LIN {X 0,Y 369.974,Z 1121.521,A -85,B 0,C 180,E1 18072.043,E2 18072.043} C_VEL
LIN {X 0,Y 371.684,Z 1112.764,A -85,B 0,C 180,E1 18068.54,E2 18068.54} C_VEL
LIN {X 0,Y 373.899,Z 1103.179,A -85,B 0,C 180,E1 18065.344,E2 18065.344} C_VEL
LIN {X 0,Y 376.935,Z 1091.306,A -85,B 0,C 180,E1 18062.045,E2 18062.045} C_VEL
LIN {X 0,Y 380.529,Z 1078.476,A -85,B 0,C 180,E1 18059.003,E2 18059.003} C_VEL
LIN {X 0,Y 384.517,Z 1064.377,A -85,B 0,C 180,E1 18056.189,E2 18056.189} C_VEL
LIN {X 0,Y 389.236,Z 1048.185,A -85,B 0,C 180,E1 18053.419,E2 18053.419} C_VEL
LIN {X 0,Y 393.672,Z 1032.569,A -85,B 0,C 180,E1 18051.146,E2 18051.146} C_VEL
LIN {X 0,Y 399.011,Z 1013.125,A -85,B 0,C 180,E1 18048.743,E2 18048.743} C_VEL
LIN {X 0,Y 403.673,Z 995.222,A -85,B 0,C 180,E1 18046.873,E2 18046.873} C_VEL
LIN {X 0,Y 408.313,Z 975.608,A -85,B 0,C 180,E1 18045.151,E2 18045.151} C_VEL
LIN {X 0,Y 412.424,Z 956.575,A -85,B 0,C 180,E1 18043.742,E2 18043.742} C_VEL
LIN {X 0,Y 416.471,Z 934.827,A -85,B 0,C 180,E1 18042.425,E2 18042.425} C_VEL
LIN {X 0,Y 419.947,Z 913.057,A -85,B 0,C 180,E1 18041.359,E2 18041.359} C_VEL
LIN {X 0,Y 422.727,Z 890.385,A -85,B 0,C 180,E1 18040.517,E2 18040.517} C_VEL
LIN {X 0,Y 424.934,Z 866.356,A -85,B 0,C 180,E1 18039.872,E2 18039.872} C_VEL
LIN {X 0,Y 433.354,Z 685.979,A -85,B 0,C 180,E1 18036.447,E2 18036.447} C_VEL
LIN {X 0,Y 436.488,Z 620.977,A -85,B 0,C 180,E1 18035.218,E2 18035.218} C_VEL
LIN {X 0,Y 425.983,Z 605.601,A -85,B 0,C 180,E1 18032.674,E2 18032.674} C_VEL
LIN {X 0,Y 417.336,Z 593.961,A -85,B 0,C 180,E1 18030.366,E2 18030.366} C_VEL
LIN {X 0,Y 410.196,Z 584.627,A -85,B 0,C 180,E1 18028.261,E2 18028.261} C_VEL
LIN {X 0,Y 406.17,Z 579.545,A -85,B 0,C 180,E1 18026.98,E2 18026.98} C_VEL
LIN {X 0,Y 402.194,Z 574.58,A -85,B 0,C 180,E1 18025.631,E2 18025.631} C_VEL
LIN {X 0,Y 398.427,Z 569.939,A -85,B 0,C 180,E1 18024.264,E2 18024.264} C_VEL
LIN {X 0,Y 393.864,Z 564.736,A -85,B 0,C 180,E1 18022.484,E2 18022.484} C_VEL
LIN {X 0,Y 392.693,Z 563.037,A -85,B 0,C 180,E1 18021.98,E2 18021.98} C_VEL
LIN {X 0,Y 389.293,Z 559.846,A -85,B 0,C 180,E1 18020.523,E2 18020.523} C_VEL
LIN {X 0,Y 387.428,Z 556.914,A -85,B 0,C 180,E1 18019.603,E2 18019.603} C_VEL
LIN {X 0,Y 384.221,Z 554.346,A -85,B 0,C 180,E1 18018.04,E2 18018.04} C_VEL
LIN {X 0,Y 382.022,Z 550.476,A -85,B 0,C 180,E1 18016.733,E2 18016.733} C_VEL
LIN {X 0,Y 378.428,Z 548.236,A -85,B 0,C 180,E1 18014.615,E2 18014.615} C_VEL
LIN {X 0,Y 376.464,Z 544.941,A -85,B 0,C 180,E1 18013.126,E2 18013.126} C_VEL
LIN {X 0,Y 376.048,Z 543.83,A -85,B 0,C 180,E1 18012.75,E2 18012.75} C_VEL
LIN {X 0,Y 372.297,Z 541.914,A -85,B 0,C 180,E1 18009.585,E2 18009.585} C_VEL
LIN {X 0,Y 370.014,Z 538.337,A -85,B 0,C 180,E1 18006.517,E2 18006.517} C_VEL
LIN {X 0,Y 369.746,Z 536.98,A -85,B 0,C 180,E1 18005.743,E2 18005.743} C_VEL
LIN {X 0,Y 369.744,Z 536.974,A -85,B 0,C 180,E1 18001.55,E2 18001.55} C_VEL
LIN {X 0,Y 369.74,Z 536.973,A -85,B 0,C 180,E1 17997.521,E2 17997.521} C_VEL
LIN {X 0,Y 369.757,Z 537.107,A -85,B 0,C 180,E1 17994.57,E2 17994.57} C_VEL
LIN {X 0,Y 370.779,Z 540.029,A -85,B 0,C 180,E1 17992.719,E2 17992.719} C_VEL
LIN {X 0,Y 373.759,Z 542.916,A -85,B 0,C 180,E1 17989.519,E2 17989.519} C_VEL
LIN {X 0,Y 376.203,Z 544.056,A -85,B 0,C 180,E1 17987.608,E2 17987.608} C_VEL
LIN {X 0,Y 377.601,Z 547.177,A -85,B 0,C 180,E1 17986.448,E2 17986.448} C_VEL
LIN {X 0,Y 380.461,Z 549.827,A -85,B 0,C 180,E1 17984.608,E2 17984.608} C_VEL
LIN {X 0,Y 382.158,Z 550.727,A -85,B 0,C 180,E1 17983.665,E2 17983.665} C_VEL
LIN {X 0,Y 384.245,Z 554.349,A -85,B 0,C 180,E1 17982.432,E2 17982.432} C_VEL
LIN {X 0,Y 387.893,Z 557.427,A -85,B 0,C 180,E1 17980.657,E2 17980.657} C_VEL
LIN {X 0,Y 390.551,Z 561.348,A -85,B 0,C 180,E1 17979.39,E2 17979.39} C_VEL
LIN {X 0,Y 393.287,Z 563.765,A -85,B 0,C 180,E1 17978.251,E2 17978.251} C_VEL
LIN {X 0,Y 396.379,Z 567.873,A -85,B 0,C 180,E1 17976.985,E2 17976.985} C_VEL
LIN {X 0,Y 398.446,Z 569.988,A -85,B 0,C 180,E1 17976.21,E2 17976.21} C_VEL
LIN {X 0,Y 406.022,Z 579.905,A -85,B 0,C 180,E1 17973.531,E2 17973.531} C_VEL
LIN {X 0,Y 413.975,Z 590.853,A -85,B 0,C 180,E1 17971.036,E2 17971.036} C_VEL
LIN {X 0,Y 422.851,Z 603.946,A -85,B 0,C 180,E1 17968.536,E2 17968.536} C_VEL
LIN {X 0,Y 431.125,Z 616.822,A -85,B 0,C 180,E1 17966.419,E2 17966.419} C_VEL
LIN {X 0,Y 436.595,Z 626.032,A -85,B 0,C 180,E1 17965.103,E2 17965.103} C_VEL
LIN {X 0,Y 426.617,Z 841.95,A -85,B 0,C 180,E1 17961.024,E2 17961.024} C_VEL
LIN {X 0,Y 424.207,Z 890.642,A -85,B 0,C 180,E1 17960.077,E2 17960.077} C_VEL
LIN {X 0,Y 421.841,Z 913.593,A -85,B 0,C 180,E1 17959.447,E2 17959.447} C_VEL
LIN {X 0,Y 418.914,Z 935.594,A -85,B 0,C 180,E1 17958.636,E2 17958.636} C_VEL
LIN {X 0,Y 415.455,Z 956.499,A -85,B 0,C 180,E1 17957.633,E2 17957.633} C_VEL
LIN {X 0,Y 411.316,Z 978.245,A -85,B 0,C 180,E1 17956.341,E2 17956.341} C_VEL
LIN {X 0,Y 407.088,Z 997.769,A -85,B 0,C 180,E1 17954.921,E2 17954.921} C_VEL
LIN {X 0,Y 402.036,Z 1019.156,A -85,B 0,C 180,E1 17953.053,E2 17953.053} C_VEL
LIN {X 0,Y 397.539,Z 1036.83,A -85,B 0,C 180,E1 17951.221,E2 17951.221} C_VEL
LIN {X 0,Y 392.445,Z 1055.81,A -85,B 0,C 180,E1 17948.904,E2 17948.904} C_VEL
LIN {X 0,Y 387.77,Z 1073.02,A -85,B 0,C 180,E1 17946.44,E2 17946.44} C_VEL
LIN {X 0,Y 383.358,Z 1088.948,A -85,B 0,C 180,E1 17943.748,E2 17943.748} C_VEL
LIN {X 0,Y 379.505,Z 1103.464,A -85,B 0,C 180,E1 17940.914,E2 17940.914} C_VEL
LIN {X 0,Y 376.133,Z 1116.554,A -85,B 0,C 180,E1 17937.895,E2 17937.895} C_VEL
LIN {X 0,Y 373.235,Z 1129.035,A -85,B 0,C 180,E1 17934.534,E2 17934.534} C_VEL
LIN {X 0,Y 371.275,Z 1138.569,A -85,B 0,C 180,E1 17931.484,E2 17931.484} C_VEL
LIN {X 0,Y 369.619,Z 1148.226,A -85,B 0,C 180,E1 17927.789,E2 17927.789} C_VEL
LIN {X 0,Y 368.729,Z 1154.956,A -85,B 0,C 180,E1 17924.606,E2 17924.606} C_VEL
LIN {X 0,Y 368.194,Z 1161.002,A -85,B 0,C 180,E1 17920.958,E2 17920.958} C_VEL
LIN {X 0,Y 367.999,Z 1164.643,A -85,B 0,C 180,E1 17917.965,E2 17917.965} C_VEL
LIN {X 0,Y 367.927,Z 1167.483,A -85,B 0,C 180,E1 17914.52,E2 17914.52} C_VEL
LIN {X 0,Y 367.923,Z 1168.636,A -85,B 0,C 180,E1 17911.245,E2 17911.245} C_VEL
LIN {X 0,Y 367.926,Z 1168.565,A -85,B 0,C 180,E1 17908.287,E2 17908.287} C_VEL
LIN {X 0,Y 367.93,Z 1167.053,A -85,B 0,C 180,E1 17904.855,E2 17904.855} C_VEL
LIN {X 0,Y 368.013,Z 1164.312,A -85,B 0,C 180,E1 17901.72,E2 17901.72} C_VEL
LIN {X 0,Y 368.272,Z 1159.89,A -85,B 0,C 180,E1 17898.251,E2 17898.251} C_VEL
LIN {X 0,Y 368.841,Z 1154.02,A -85,B 0,C 180,E1 17894.915,E2 17894.915} C_VEL
LIN {X 0,Y 369.869,Z 1146.741,A -85,B 0,C 180,E1 17891.561,E2 17891.561} C_VEL
LIN {X 0,Y 371.46,Z 1137.631,A -85,B 0,C 180,E1 17888.194,E2 17888.194} C_VEL
LIN {X 0,Y 373.736,Z 1126.85,A -85,B 0,C 180,E1 17884.825,E2 17884.825} C_VEL
LIN {X 0,Y 376.617,Z 1114.607,A -85,B 0,C 180,E1 17881.626,E2 17881.626} C_VEL
LIN {X 0,Y 380.345,Z 1100.097,A -85,B 0,C 180,E1 17878.4,E2 17878.4} C_VEL
LIN {X 0,Y 384.323,Z 1085.496,A -85,B 0,C 180,E1 17875.628,E2 17875.628} C_VEL
LIN {X 0,Y 388.891,Z 1068.742,A -85,B 0,C 180,E1 17872.921,E2 17872.921} C_VEL
LIN {X 0,Y 393.728,Z 1051.242,A -85,B 0,C 180,E1 17870.495,E2 17870.495} C_VEL
LIN {X 0,Y 398.569,Z 1032.731,A -85,B 0,C 180,E1 17868.334,E2 17868.334} C_VEL
LIN {X 0,Y 403.725,Z 1012.106,A -85,B 0,C 180,E1 17866.293,E2 17866.293} C_VEL
LIN {X 0,Y 408.111,Z 993.164,A -85,B 0,C 180,E1 17864.724,E2 17864.724} C_VEL
LIN {X 0,Y 412.553,Z 971.99,A -85,B 0,C 180,E1 17863.266,E2 17863.266} C_VEL
LIN {X 0,Y 416.147,Z 952.514,A -85,B 0,C 180,E1 17862.164,E2 17862.164} C_VEL
LIN {X 0,Y 419.778,Z 929.35,A -85,B 0,C 180,E1 17861.118,E2 17861.118} C_VEL
LIN {X 0,Y 422.268,Z 909.791,A -85,B 0,C 180,E1 17860.439,E2 17860.439} C_VEL
LIN {X 0,Y 424.551,Z 884.65,A -85,B 0,C 180,E1 17859.8,E2 17859.8} C_VEL
LIN {X 0,Y 433.122,Z 697.721,A -85,B 0,C 180,E1 17856.257,E2 17856.257} C_VEL
LIN {X 0,Y 436.44,Z 625.581,A -85,B 0,C 180,E1 17854.869,E2 17854.869} C_VEL
LIN {X 0,Y 425.319,Z 607.642,A -85,B 0,C 180,E1 17852.132,E2 17852.132} C_VEL
LIN {X 0,Y 415.18,Z 592.599,A -85,B 0,C 180,E1 17849.345,E2 17849.345} C_VEL
LIN {X 0,Y 407.907,Z 582.585,A -85,B 0,C 180,E1 17847.124,E2 17847.124} C_VEL
LIN {X 0,Y 403.893,Z 577.15,A -85,B 0,C 180,E1 17845.79,E2 17845.79} C_VEL
LIN {X 0,Y 400.129,Z 572.41,A -85,B 0,C 180,E1 17844.467,E2 17844.467} C_VEL
LIN {X 0,Y 397.545,Z 568.885,A -85,B 0,C 180,E1 17843.493,E2 17843.493} C_VEL
LIN {X 0,Y 394.054,Z 565.064,A -85,B 0,C 180,E1 17842.135,E2 17842.135} C_VEL
LIN {X 0,Y 392.77,Z 563.107,A -85,B 0,C 180,E1 17841.582,E2 17841.582} C_VEL
LIN {X 0,Y 389.424,Z 560.029,A -85,B 0,C 180,E1 17840.163,E2 17840.163} C_VEL
LIN {X 0,Y 387.637,Z 556.986,A -85,B 0,C 180,E1 17839.278,E2 17839.278} C_VEL
LIN {X 0,Y 384.248,Z 554.358,A -85,B 0,C 180,E1 17837.646,E2 17837.646} C_VEL
LIN {X 0,Y 382.144,Z 550.727,A -85,B 0,C 180,E1 17836.414,E2 17836.414} C_VEL
LIN {X 0,Y 378.187,Z 547.968,A -85,B 0,C 180,E1 17834.077,E2 17834.077} C_VEL
LIN {X 0,Y 376.387,Z 544.727,A -85,B 0,C 180,E1 17832.698,E2 17832.698} C_VEL
LIN {X 0,Y 376.11,Z 543.795,A -85,B 0,C 180,E1 17832.435,E2 17832.435} C_VEL
LIN {X 0,Y 372.136,Z 541.73,A -85,B 0,C 180,E1 17829.121,E2 17829.121} C_VEL
LIN {X 0,Y 370.12,Z 538.604,A -85,B 0,C 180,E1 17826.514,E2 17826.514} C_VEL
LIN {X 0,Y 369.739,Z 536.974,A -85,B 0,C 180,E1 17825.586,E2 17825.586} C_VEL
LIN {X 0,Y 369.738,Z 536.977,A -85,B 0,C 180,E1 17821.394,E2 17821.394} C_VEL
LIN {X 0,Y 369.729,Z 536.982,A -85,B 0,C 180,E1 17817.365,E2 17817.365} C_VEL
LIN {X 0,Y 369.766,Z 537.211,A -85,B 0,C 180,E1 17813.634,E2 17813.634} C_VEL
LIN {X 0,Y 370.756,Z 539.978,A -85,B 0,C 180,E1 17811.938,E2 17811.938} C_VEL
LIN {X 0,Y 373.997,Z 543.047,A -85,B 0,C 180,E1 17808.589,E2 17808.589} C_VEL
LIN {X 0,Y 376.203,Z 544.103,A -85,B 0,C 180,E1 17806.904,E2 17806.904} C_VEL
LIN {X 0,Y 377.726,Z 547.39,A -85,B 0,C 180,E1 17805.67,E2 17805.67} C_VEL
LIN {X 0,Y 380.657,Z 549.896,A -85,B 0,C 180,E1 17803.833,E2 17803.833} C_VEL
LIN {X 0,Y 382.168,Z 550.759,A -85,B 0,C 180,E1 17803,E2 17803} C_VEL
LIN {X 0,Y 384.353,Z 554.514,A -85,B 0,C 180,E1 17801.723,E2 17801.723} C_VEL
LIN {X 0,Y 387.868,Z 557.472,A -85,B 0,C 180,E1 17800.028,E2 17800.028} C_VEL
LIN {X 0,Y 390.55,Z 561.329,A -85,B 0,C 180,E1 17798.761,E2 17798.761} C_VEL
LIN {X 0,Y 393.217,Z 563.653,A -85,B 0,C 180,E1 17797.657,E2 17797.657} C_VEL
LIN {X 0,Y 396.404,Z 567.901,A -85,B 0,C 180,E1 17796.356,E2 17796.356} C_VEL
LIN {X 0,Y 398.392,Z 569.905,A -85,B 0,C 180,E1 17795.616,E2 17795.616} C_VEL
LIN {X 0,Y 402.071,Z 574.487,A -85,B 0,C 180,E1 17794.282,E2 17794.282} C_VEL
LIN {X 0,Y 403.96,Z 576.86,A -85,B 0,C 180,E1 17793.63,E2 17793.63} C_VEL
LIN {X 0,Y 408.347,Z 582.296,A -85,B 0,C 180,E1 17792.196,E2 17792.196} C_VEL
LIN {X 0,Y 412.91,Z 588.21,A -85,B 0,C 180,E1 17790.795,E2 17790.795} C_VEL
LIN {X 0,Y 420.03,Z 597.504,A -85,B 0,C 180,E1 17788.779,E2 17788.779} C_VEL
LIN {X 0,Y 430.409,Z 611.995,A -85,B 0,C 180,E1 17786.115,E2 17786.115} C_VEL
LIN {X 0,Y 436.464,Z 621.114,A -85,B 0,C 180,E1 17784.679,E2 17784.679} C_VEL
LIN {X 0,Y 426.709,Z 829.94,A -85,B 0,C 180,E1 17780.74,E2 17780.74} C_VEL
LIN {X 0,Y 424.596,Z 870.779,A -85,B 0,C 180,E1 17779.937,E2 17779.937} C_VEL
LIN {X 0,Y 422.391,Z 893.197,A -85,B 0,C 180,E1 17779.296,E2 17779.296} C_VEL
LIN {X 0,Y 419.347,Z 916.813,A -85,B 0,C 180,E1 17778.374,E2 17778.374} C_VEL
LIN {X 0,Y 416.239,Z 936.052,A -85,B 0,C 180,E1 17777.414,E2 17777.414} C_VEL
LIN {X 0,Y 411.993,Z 958.492,A -85,B 0,C 180,E1 17776.03,E2 17776.03} C_VEL
LIN {X 0,Y 408.091,Z 976.509,A -85,B 0,C 180,E1 17774.683,E2 17774.683} C_VEL
LIN {X 0,Y 403.076,Z 997.396,A -85,B 0,C 180,E1 17772.819,E2 17772.819} C_VEL
LIN {X 0,Y 398.419,Z 1015.308,A -85,B 0,C 180,E1 17770.92,E2 17770.92} C_VEL
LIN {X 0,Y 393.512,Z 1033.103,A -85,B 0,C 180,E1 17768.687,E2 17768.687} C_VEL
LIN {X 0,Y 388.822,Z 1049.667,A -85,B 0,C 180,E1 17766.26,E2 17766.26} C_VEL
LIN {X 0,Y 384.391,Z 1064.772,A -85,B 0,C 180,E1 17763.646,E2 17763.646} C_VEL
LIN {X 0,Y 380.431,Z 1078.817,A -85,B 0,C 180,E1 17760.831,E2 17760.831} C_VEL
LIN {X 0,Y 378.216,Z 1086.719,A -85,B 0,C 180,E1 17759.02,E2 17759.02} C_VEL
LIN {X 0,Y 376.201,Z 1090.945,A -85,B 0,C 180,E1 17758.078,E2 17758.078} C_VEL
LIN {X 0,Y 367.563,Z 1101.74,A -85,B 0,C 180,E1 17755.588,E2 17755.588} C_VEL
LIN {X 0,Y 366.052,Z 1104.763,A -85,B 0,C 180,E1 17754.692,E2 17754.692} C_VEL
LIN {X 0,Y 363.781,Z 1114.173,A -85,B 0,C 180,E1 17751.442,E2 17751.442} C_VEL
LIN {X 0,Y 362.006,Z 1122.695,A -85,B 0,C 180,E1 17747.854,E2 17747.854} C_VEL
LIN {X 0,Y 360.934,Z 1129.295,A -85,B 0,C 180,E1 17744.438,E2 17744.438} C_VEL
LIN {X 0,Y 360.309,Z 1134.534,A -85,B 0,C 180,E1 17740.877,E2 17740.877} C_VEL
LIN {X 0,Y 360.035,Z 1138.029,A -85,B 0,C 180,E1 17737.661,E2 17737.661} C_VEL
LIN {X 0,Y 359.946,Z 1140.516,A -85,B 0,C 180,E1 17733.982,E2 17733.982} C_VEL
LIN {X 0,Y 359.922,Z 1141.386,A -85,B 0,C 180,E1 17730.955,E2 17730.955} C_VEL
LIN {X 0,Y 359.937,Z 1141.148,A -85,B 0,C 180,E1 17727.453,E2 17727.453} C_VEL
LIN {X 0,Y 359.967,Z 1139.462,A -85,B 0,C 180,E1 17724.101,E2 17724.101} C_VEL
LIN {X 0,Y 360.154,Z 1136.572,A -85,B 0,C 180,E1 17720.734,E2 17720.734} C_VEL
LIN {X 0,Y 360.579,Z 1131.982,A -85,B 0,C 180,E1 17717.183,E2 17717.183} C_VEL
LIN {X 0,Y 361.415,Z 1126.219,A -85,B 0,C 180,E1 17713.775,E2 17713.775} C_VEL
LIN {X 0,Y 362.854,Z 1118.465,A -85,B 0,C 180,E1 17710.188,E2 17710.188} C_VEL
LIN {X 0,Y 364.909,Z 1109.488,A -85,B 0,C 180,E1 17706.761,E2 17706.761} C_VEL
LIN {X 0,Y 367.708,Z 1098.548,A -85,B 0,C 180,E1 17703.342,E2 17703.342} C_VEL
LIN {X 0,Y 371.189,Z 1086.365,A -85,B 0,C 180,E1 17700.111,E2 17700.111} C_VEL
LIN {X 0,Y 374.999,Z 1073.488,A -85,B 0,C 180,E1 17697.231,E2 17697.231} C_VEL
LIN {X 0,Y 379.793,Z 1057.789,A -85,B 0,C 180,E1 17694.236,E2 17694.236} C_VEL
LIN {X 0,Y 384.442,Z 1042.497,A -85,B 0,C 180,E1 17691.758,E2 17691.758} C_VEL
LIN {X 0,Y 389.665,Z 1024.824,A -85,B 0,C 180,E1 17689.326,E2 17689.326} C_VEL
LIN {X 0,Y 394.549,Z 1007.564,A -85,B 0,C 180,E1 17687.3,E2 17687.3} C_VEL
LIN {X 0,Y 399.514,Z 988.481,A -85,B 0,C 180,E1 17685.412,E2 17685.412} C_VEL
LIN {X 0,Y 404.278,Z 968.766,A -85,B 0,C 180,E1 17683.766,E2 17683.766} C_VEL
LIN {X 0,Y 408.611,Z 948.141,A -85,B 0,C 180,E1 17682.355,E2 17682.355} C_VEL
LIN {X 0,Y 412.602,Z 926.618,A -85,B 0,C 180,E1 17681.146,E2 17681.146} C_VEL
LIN {X 0,Y 415.736,Z 905.591,A -85,B 0,C 180,E1 17680.218,E2 17680.218} C_VEL
LIN {X 0,Y 418.471,Z 882.758,A -85,B 0,C 180,E1 17679.442,E2 17679.442} C_VEL
LIN {X 0,Y 420.221,Z 860.799,A -85,B 0,C 180,E1 17678.912,E2 17678.912} C_VEL
LIN {X 0,Y 429.901,Z 661.299,A -85,B 0,C 180,E1 17675.114,E2 17675.114} C_VEL
LIN {X 0,Y 431.671,Z 625.138,A -85,B 0,C 180,E1 17674.414,E2 17674.414} C_VEL
LIN {X 0,Y 422.321,Z 611.429,A -85,B 0,C 180,E1 17672.068,E2 17672.068} C_VEL
LIN {X 0,Y 414.179,Z 600.251,A -85,B 0,C 180,E1 17669.822,E2 17669.822} C_VEL
LIN {X 0,Y 407.276,Z 591.159,A -85,B 0,C 180,E1 17667.725,E2 17667.725} C_VEL
LIN {X 0,Y 403.607,Z 586.459,A -85,B 0,C 180,E1 17666.522,E2 17666.522} C_VEL
LIN {X 0,Y 399.717,Z 581.583,A -85,B 0,C 180,E1 17665.166,E2 17665.166} C_VEL
LIN {X 0,Y 395.235,Z 576.057,A -85,B 0,C 180,E1 17663.481,E2 17663.481} C_VEL
LIN {X 0,Y 391.616,Z 571.678,A -85,B 0,C 180,E1 17662.005,E2 17662.005} C_VEL
LIN {X 0,Y 390.571,Z 570.382,A -85,B 0,C 180,E1 17661.553,E2 17661.553} C_VEL
LIN {X 0,Y 387.196,Z 566.895,A -85,B 0,C 180,E1 17660.048,E2 17660.048} C_VEL
LIN {X 0,Y 385.874,Z 564.637,A -85,B 0,C 180,E1 17659.37,E2 17659.37} C_VEL
LIN {X 0,Y 382.582,Z 561.89,A -85,B 0,C 180,E1 17657.726,E2 17657.726} C_VEL
LIN {X 0,Y 380.276,Z 558.156,A -85,B 0,C 180,E1 17656.34,E2 17656.34} C_VEL
LIN {X 0,Y 376.808,Z 555.68,A -85,B 0,C 180,E1 17654.209,E2 17654.209} C_VEL
LIN {X 0,Y 374.843,Z 552.084,A -85,B 0,C 180,E1 17652.635,E2 17652.635} C_VEL
LIN {X 0,Y 374.274,Z 551.558,A -85,B 0,C 180,E1 17652.184,E2 17652.184} C_VEL
LIN {X 0,Y 370.628,Z 549.247,A -85,B 0,C 180,E1 17648.846,E2 17648.846} C_VEL
LIN {X 0,Y 368.792,Z 545.751,A -85,B 0,C 180,E1 17646.07,E2 17646.07} C_VEL
LIN {X 0,Y 368.514,Z 544.882,A -85,B 0,C 180,E1 17645.45,E2 17645.45} C_VEL
LIN {X 0,Y 367.489,Z 544.65,A -85,B 0,C 180,E1 17637.349,E2 17637.349} C_VEL
LIN {X 0,Y 368.674,Z 545.169,A -85,B 0,C 180,E1 17634.71,E2 17634.71} C_VEL
LIN {X 0,Y 370.02,Z 548.462,A -85,B 0,C 180,E1 17632.392,E2 17632.392} C_VEL
LIN {X 0,Y 373.522,Z 551.238,A -85,B 0,C 180,E1 17628.888,E2 17628.888} C_VEL
LIN {X 0,Y 374.781,Z 551.857,A -85,B 0,C 180,E1 17627.912,E2 17627.912} C_VEL
LIN {X 0,Y 376.512,Z 555.301,A -85,B 0,C 180,E1 17626.486,E2 17626.486} C_VEL
LIN {X 0,Y 379.513,Z 557.837,A -85,B 0,C 180,E1 17624.569,E2 17624.569} C_VEL
LIN {X 0,Y 380.599,Z 558.552,A -85,B 0,C 180,E1 17623.949,E2 17623.949} C_VEL
LIN {X 0,Y 383.003,Z 562.351,A -85,B 0,C 180,E1 17622.53,E2 17622.53} C_VEL
LIN {X 0,Y 386.169,Z 565.122,A -85,B 0,C 180,E1 17620.96,E2 17620.96} C_VEL
LIN {X 0,Y 388.957,Z 569.05,A -85,B 0,C 180,E1 17619.616,E2 17619.616} C_VEL
LIN {X 0,Y 391.401,Z 571.327,A -85,B 0,C 180,E1 17618.574,E2 17618.574} C_VEL
LIN {X 0,Y 394.72,Z 575.585,A -85,B 0,C 180,E1 17617.198,E2 17617.198} C_VEL
LIN {X 0,Y 396.397,Z 577.418,A -85,B 0,C 180,E1 17616.553,E2 17616.553} C_VEL
LIN {X 0,Y 403.575,Z 586.93,A -85,B 0,C 180,E1 17613.952,E2 17613.952} C_VEL
LIN {X 0,Y 411.399,Z 597.894,A -85,B 0,C 180,E1 17611.434,E2 17611.434} C_VEL
LIN {X 0,Y 419.924,Z 610.688,A -85,B 0,C 180,E1 17608.97,E2 17608.97} C_VEL
LIN {X 0,Y 427.959,Z 623.406,A -85,B 0,C 180,E1 17606.859,E2 17606.859} C_VEL
LIN {X 0,Y 431.824,Z 630.006,A -85,B 0,C 180,E1 17605.898,E2 17605.898} C_VEL
LIN {X 0,Y 421.453,Z 844.861,A -85,B 0,C 180,E1 17601.814,E2 17601.814} C_VEL
LIN {X 0,Y 419.072,Z 890.519,A -85,B 0,C 180,E1 17600.917,E2 17600.917} C_VEL
LIN {X 0,Y 416.645,Z 913.302,A -85,B 0,C 180,E1 17600.289,E2 17600.289} C_VEL
LIN {X 0,Y 413.637,Z 935.155,A -85,B 0,C 180,E1 17599.484,E2 17599.484} C_VEL
LIN {X 0,Y 410.022,Z 956.201,A -85,B 0,C 180,E1 17598.472,E2 17598.472} C_VEL
LIN {X 0,Y 405.661,Z 978.179,A -85,B 0,C 180,E1 17597.161,E2 17597.161} C_VEL
LIN {X 0,Y 401.099,Z 998.374,A -85,B 0,C 180,E1 17595.679,E2 17595.679} C_VEL
LIN {X 0,Y 395.834,Z 1019.592,A -85,B 0,C 180,E1 17593.797,E2 17593.797} C_VEL
LIN {X 0,Y 390.974,Z 1037.873,A -85,B 0,C 180,E1 17591.872,E2 17591.872} C_VEL
LIN {X 0,Y 385.827,Z 1056.062,A -85,B 0,C 180,E1 17589.606,E2 17589.606} C_VEL
LIN {X 0,Y 380.958,Z 1073.08,A -85,B 0,C 180,E1 17587.132,E2 17587.132} C_VEL
LIN {X 0,Y 376.414,Z 1088.635,A -85,B 0,C 180,E1 17584.457,E2 17584.457} C_VEL
LIN {X 0,Y 372.316,Z 1103.15,A -85,B 0,C 180,E1 17581.579,E2 17581.579} C_VEL
LIN {X 0,Y 368.742,Z 1116.241,A -85,B 0,C 180,E1 17578.504,E2 17578.504} C_VEL
LIN {X 0,Y 365.653,Z 1128.722,A -85,B 0,C 180,E1 17575.077,E2 17575.077} C_VEL
LIN {X 0,Y 363.455,Z 1138.728,A -85,B 0,C 180,E1 17571.801,E2 17571.801} C_VEL
LIN {X 0,Y 361.703,Z 1148.276,A -85,B 0,C 180,E1 17568.027,E2 17568.027} C_VEL
LIN {X 0,Y 360.764,Z 1154.96,A -85,B 0,C 180,E1 17564.772,E2 17564.772} C_VEL
LIN {X 0,Y 360.202,Z 1160.911,A -85,B 0,C 180,E1 17561.042,E2 17561.042} C_VEL
LIN {X 0,Y 359.985,Z 1164.669,A -85,B 0,C 180,E1 17557.822,E2 17557.822} C_VEL
LIN {X 0,Y 359.933,Z 1167.349,A -85,B 0,C 180,E1 17554.245,E2 17554.245} C_VEL
LIN {X 0,Y 359.929,Z 1168.337,A -85,B 0,C 180,E1 17551.273,E2 17551.273} C_VEL
LIN {X 0,Y 359.931,Z 1168.266,A -85,B 0,C 180,E1 17548.249,E2 17548.249} C_VEL
LIN {X 0,Y 359.931,Z 1166.752,A -85,B 0,C 180,E1 17544.74,E2 17544.74} C_VEL
LIN {X 0,Y 360.021,Z 1164.009,A -85,B 0,C 180,E1 17541.535,E2 17541.535} C_VEL
LIN {X 0,Y 360.304,Z 1159.585,A -85,B 0,C 180,E1 17537.987,E2 17537.987} C_VEL
LIN {X 0,Y 360.922,Z 1153.712,A -85,B 0,C 180,E1 17534.576,E2 17534.576} C_VEL
LIN {X 0,Y 362.032,Z 1146.43,A -85,B 0,C 180,E1 17531.147,E2 17531.147} C_VEL
LIN {X 0,Y 363.739,Z 1137.318,A -85,B 0,C 180,E1 17527.707,E2 17527.707} C_VEL
LIN {X 0,Y 366.177,Z 1126.535,A -85,B 0,C 180,E1 17524.268,E2 17524.268} C_VEL
LIN {X 0,Y 369.082,Z 1114.939,A -85,B 0,C 180,E1 17521.17,E2 17521.17} C_VEL
LIN {X 0,Y 372.995,Z 1100.606,A -85,B 0,C 180,E1 17517.894,E2 17517.894} C_VEL
LIN {X 0,Y 377.168,Z 1086.038,A -85,B 0,C 180,E1 17515.067,E2 17515.067} C_VEL
LIN {X 0,Y 382.104,Z 1068.94,A -85,B 0,C 180,E1 17512.242,E2 17512.242} C_VEL
LIN {X 0,Y 387.167,Z 1051.524,A -85,B 0,C 180,E1 17509.787,E2 17509.787} C_VEL
LIN {X 0,Y 392.269,Z 1032.909,A -85,B 0,C 180,E1 17507.582,E2 17507.582} C_VEL
LIN {X 0,Y 397.461,Z 1013.196,A -85,B 0,C 180,E1 17505.596,E2 17505.596} C_VEL
LIN {X 0,Y 402.161,Z 993.759,A -85,B 0,C 180,E1 17503.965,E2 17503.965} C_VEL
LIN {X 0,Y 407.023,Z 971.569,A -85,B 0,C 180,E1 17502.422,E2 17502.422} C_VEL
LIN {X 0,Y 410.735,Z 952.202,A -85,B 0,C 180,E1 17501.323,E2 17501.323} C_VEL
LIN {X 0,Y 414.5,Z 929.035,A -85,B 0,C 180,E1 17500.275,E2 17500.275} C_VEL
LIN {X 0,Y 417.114,Z 909.231,A -85,B 0,C 180,E1 17499.589,E2 17499.589} C_VEL
LIN {X 0,Y 419.451,Z 884.222,A -85,B 0,C 180,E1 17498.953,E2 17498.953} C_VEL
LIN {X 0,Y 428.475,Z 696.003,A -85,B 0,C 180,E1 17495.361,E2 17495.361} C_VEL
LIN {X 0,Y 431.66,Z 629.576,A -85,B 0,C 180,E1 17494.073,E2 17494.073} C_VEL
LIN {X 0,Y 421.435,Z 613.049,A -85,B 0,C 180,E1 17491.463,E2 17491.463} C_VEL
LIN {X 0,Y 412.16,Z 599.033,A -85,B 0,C 180,E1 17488.825,E2 17488.825} C_VEL
LIN {X 0,Y 405.128,Z 589.212,A -85,B 0,C 180,E1 17486.611,E2 17486.611} C_VEL
LIN {X 0,Y 401.196,Z 583.811,A -85,B 0,C 180,E1 17485.263,E2 17485.263} C_VEL
LIN {X 0,Y 395.328,Z 576.131,A -85,B 0,C 180,E1 17483.08,E2 17483.08} C_VEL
LIN {X 0,Y 391.76,Z 571.952,A -85,B 0,C 180,E1 17481.641,E2 17481.641} C_VEL
LIN {X 0,Y 390.638,Z 570.462,A -85,B 0,C 180,E1 17481.155,E2 17481.155} C_VEL
LIN {X 0,Y 387.242,Z 566.97,A -85,B 0,C 180,E1 17479.652,E2 17479.652} C_VEL
LIN {X 0,Y 385.765,Z 564.546,A -85,B 0,C 180,E1 17478.904,E2 17478.904} C_VEL
LIN {X 0,Y 382.339,Z 561.569,A -85,B 0,C 180,E1 17477.188,E2 17477.188} C_VEL
LIN {X 0,Y 380.409,Z 558.216,A -85,B 0,C 180,E1 17476.02,E2 17476.02} C_VEL
LIN {X 0,Y 376.995,Z 555.899,A -85,B 0,C 180,E1 17473.966,E2 17473.966} C_VEL
LIN {X 0,Y 374.962,Z 552.454,A -85,B 0,C 180,E1 17472.395,E2 17472.395} C_VEL
LIN {X 0,Y 374.525,Z 551.588,A -85,B 0,C 180,E1 17472.018,E2 17472.018} C_VEL
LIN {X 0,Y 370.736,Z 549.325,A -85,B 0,C 180,E1 17468.686,E2 17468.686} C_VEL
LIN {X 0,Y 368.871,Z 546.024,A -85,B 0,C 180,E1 17466.068,E2 17466.068} C_VEL
LIN {X 0,Y 368.588,Z 544.891,A -85,B 0,C 180,E1 17465.448,E2 17465.448} C_VEL
LIN {X 0,Y 367.101,Z 544.538,A -85,B 0,C 180,E1 17457.346,E2 17457.346} C_VEL
LIN {X 0,Y 368.644,Z 545.132,A -85,B 0,C 180,E1 17453.85,E2 17453.85} C_VEL
LIN {X 0,Y 370.005,Z 548.429,A -85,B 0,C 180,E1 17451.609,E2 17451.609} C_VEL
LIN {X 0,Y 373.599,Z 551.273,A -85,B 0,C 180,E1 17448.107,E2 17448.107} C_VEL
LIN {X 0,Y 374.777,Z 551.897,A -85,B 0,C 180,E1 17447.206,E2 17447.206} C_VEL
LIN {X 0,Y 376.641,Z 555.498,A -85,B 0,C 180,E1 17445.706,E2 17445.706} C_VEL
LIN {X 0,Y 379.973,Z 558.03,A -85,B 0,C 180,E1 17443.646,E2 17443.646} C_VEL
LIN {X 0,Y 380.663,Z 558.708,A -85,B 0,C 180,E1 17443.245,E2 17443.245} C_VEL
LIN {X 0,Y 383.098,Z 562.5,A -85,B 0,C 180,E1 17441.827,E2 17441.827} C_VEL
LIN {X 0,Y 386.076,Z 565.033,A -85,B 0,C 180,E1 17440.365,E2 17440.365} C_VEL
LIN {X 0,Y 388.956,Z 569.03,A -85,B 0,C 180,E1 17438.985,E2 17438.985} C_VEL
LIN {X 0,Y 391.331,Z 571.22,A -85,B 0,C 180,E1 17437.979,E2 17437.979} C_VEL
LIN {X 0,Y 394.746,Z 575.619,A -85,B 0,C 180,E1 17436.567,E2 17436.567} C_VEL
LIN {X 0,Y 396.434,Z 577.488,A -85,B 0,C 180,E1 17435.921,E2 17435.921} C_VEL
LIN {X 0,Y 400.36,Z 582.21,A -85,B 0,C 180,E1 17434.481,E2 17434.481} C_VEL
LIN {X 0,Y 406.459,Z 590.135,A -85,B 0,C 180,E1 17432.414,E2 17432.414} C_VEL
LIN {X 0,Y 413.12,Z 598.758,A -85,B 0,C 180,E1 17430.374,E2 17430.374} C_VEL
LIN {X 0,Y 422.929,Z 612.268,A -85,B 0,C 180,E1 17427.664,E2 17427.664} C_VEL
LIN {X 0,Y 431.691,Z 625.297,A -85,B 0,C 180,E1 17425.472,E2 17425.472} C_VEL
LIN {X 0,Y 421.539,Z 833.534,A -85,B 0,C 180,E1 17421.52,E2 17421.52} C_VEL
LIN {X 0,Y 419.46,Z 871.421,A -85,B 0,C 180,E1 17420.765,E2 17420.765} C_VEL
LIN {X 0,Y 417.193,Z 893.642,A -85,B 0,C 180,E1 17420.126,E2 17420.126} C_VEL
LIN {X 0,Y 414.05,Z 917.125,A -85,B 0,C 180,E1 17419.206,E2 17419.206} C_VEL
LIN {X 0,Y 410.826,Z 936.364,A -85,B 0,C 180,E1 17418.242,E2 17418.242} C_VEL
LIN {X 0,Y 406.402,Z 958.87,A -85,B 0,C 180,E1 17416.846,E2 17416.846} C_VEL
LIN {X 0,Y 402.357,Z 976.82,A -85,B 0,C 180,E1 17415.496,E2 17415.496} C_VEL
LIN {X 0,Y 397.138,Z 997.707,A -85,B 0,C 180,E1 17413.618,E2 17413.618} C_VEL
LIN {X 0,Y 392.275,Z 1015.62,A -85,B 0,C 180,E1 17411.703,E2 17411.703} C_VEL
LIN {X 0,Y 386.978,Z 1033.908,A -85,B 0,C 180,E1 17409.379,E2 17409.379} C_VEL
LIN {X 0,Y 382.063,Z 1050.474,A -85,B 0,C 180,E1 17406.914,E2 17406.914} C_VEL
LIN {X 0,Y 377.286,Z 1065.916,A -85,B 0,C 180,E1 17404.183,E2 17404.183} C_VEL
LIN {X 0,Y 372.913,Z 1080.507,A -85,B 0,C 180,E1 17401.164,E2 17401.164} C_VEL
LIN {X 0,Y 369.43,Z 1092.359,A -85,B 0,C 180,E1 17398.271,E2 17398.271} C_VEL
LIN {X 0,Y 366.052,Z 1104.763,A -85,B 0,C 180,E1 17394.692,E2 17394.692} C_VEL
LIN {X 0,Y 364.246,Z 1108.282,A -85,B 0,C 180,E1 17393.635,E2 17393.635} C_VEL
LIN {X 0,Y 356.245,Z 1117.083,A -85,B 0,C 180,E1 17390.835,E2 17390.835} C_VEL
LIN {X 0,Y 354.967,Z 1119.504,A -85,B 0,C 180,E1 17389.86,E2 17389.86} C_VEL
LIN {X 0,Y 353.43,Z 1127.245,A -85,B 0,C 180,E1 17386.096,E2 17386.096} C_VEL
LIN {X 0,Y 352.6,Z 1132.738,A -85,B 0,C 180,E1 17382.715,E2 17382.715} C_VEL
LIN {X 0,Y 352.139,Z 1137.404,A -85,B 0,C 180,E1 17378.82,E2 17378.82} C_VEL
LIN {X 0,Y 351.971,Z 1140.03,A -85,B 0,C 180,E1 17375.543,E2 17375.543} C_VEL
LIN {X 0,Y 351.94,Z 1141.556,A -85,B 0,C 180,E1 17371.954,E2 17371.954} C_VEL
LIN {X 0,Y 351.934,Z 1141.655,A -85,B 0,C 180,E1 17368.698,E2 17368.698} C_VEL
LIN {X 0,Y 351.96,Z 1140.593,A -85,B 0,C 180,E1 17365.275,E2 17365.275} C_VEL
LIN {X 0,Y 352.103,Z 1137.954,A -85,B 0,C 180,E1 17361.673,E2 17361.673} C_VEL
LIN {X 0,Y 352.442,Z 1134.15,A -85,B 0,C 180,E1 17358.214,E2 17358.214} C_VEL
LIN {X 0,Y 353.197,Z 1128.585,A -85,B 0,C 180,E1 17354.568,E2 17354.568} C_VEL
LIN {X 0,Y 354.397,Z 1122.161,A -85,B 0,C 180,E1 17351.239,E2 17351.239} C_VEL
LIN {X 0,Y 356.398,Z 1113.378,A -85,B 0,C 180,E1 17347.571,E2 17347.571} C_VEL
LIN {X 0,Y 359.108,Z 1103.264,A -85,B 0,C 180,E1 17344.07,E2 17344.07} C_VEL
LIN {X 0,Y 362.44,Z 1091.749,A -85,B 0,C 180,E1 17340.772,E2 17340.772} C_VEL
LIN {X 0,Y 366.425,Z 1079.092,A -85,B 0,C 180,E1 17337.668,E2 17337.668} C_VEL
LIN {X 0,Y 370.904,Z 1064.983,A -85,B 0,C 180,E1 17334.767,E2 17334.767} C_VEL
LIN {X 0,Y 376.115,Z 1048.796,A -85,B 0,C 180,E1 17331.921,E2 17331.921} C_VEL
LIN {X 0,Y 381.149,Z 1032.721,A -85,B 0,C 180,E1 17329.531,E2 17329.531} C_VEL
LIN {X 0,Y 386.803,Z 1013.944,A -85,B 0,C 180,E1 17327.169,E2 17327.169} C_VEL
LIN {X 0,Y 391.726,Z 996.55,A -85,B 0,C 180,E1 17325.316,E2 17325.316} C_VEL
LIN {X 0,Y 396.959,Z 976.204,A -85,B 0,C 180,E1 17323.497,E2 17323.497} C_VEL
LIN {X 0,Y 401.628,Z 956.172,A -85,B 0,C 180,E1 17322.002,E2 17322.002} C_VEL
LIN {X 0,Y 405.781,Z 935.329,A -85,B 0,C 180,E1 17320.739,E2 17320.739} C_VEL
LIN {X 0,Y 409.547,Z 913.327,A -85,B 0,C 180,E1 17319.658,E2 17319.658} C_VEL
LIN {X 0,Y 412.525,Z 890.697,A -85,B 0,C 180,E1 17318.816,E2 17318.816} C_VEL
LIN {X 0,Y 414.905,Z 866.16,A -85,B 0,C 180,E1 17318.16,E2 17318.16} C_VEL
LIN {X 0,Y 424.226,Z 682.875,A -85,B 0,C 180,E1 17314.637,E2 17314.637} C_VEL
LIN {X 0,Y 426.942,Z 629.421,A -85,B 0,C 180,E1 17313.596,E2 17313.596} C_VEL
LIN {X 0,Y 418.823,Z 617.382,A -85,B 0,C 180,E1 17311.482,E2 17311.482} C_VEL
LIN {X 0,Y 409.914,Z 604.853,A -85,B 0,C 180,E1 17308.919,E2 17308.919} C_VEL
LIN {X 0,Y 401.574,Z 593.934,A -85,B 0,C 180,E1 17306.229,E2 17306.229} C_VEL
LIN {X 0,Y 397.454,Z 588.758,A -85,B 0,C 180,E1 17304.763,E2 17304.763} C_VEL
LIN {X 0,Y 393.227,Z 583.442,A -85,B 0,C 180,E1 17303.132,E2 17303.132} C_VEL
LIN {X 0,Y 389.516,Z 578.823,A -85,B 0,C 180,E1 17301.575,E2 17301.575} C_VEL
LIN {X 0,Y 385.057,Z 573.827,A -85,B 0,C 180,E1 17299.531,E2 17299.531} C_VEL
LIN {X 0,Y 384.026,Z 572.178,A -85,B 0,C 180,E1 17298.993,E2 17298.993} C_VEL
LIN {X 0,Y 380.7,Z 569.096,A -85,B 0,C 180,E1 17297.265,E2 17297.265} C_VEL
LIN {X 0,Y 378.81,Z 565.92,A -85,B 0,C 180,E1 17296.09,E2 17296.09} C_VEL
LIN {X 0,Y 375.414,Z 563.37,A -85,B 0,C 180,E1 17293.948,E2 17293.948} C_VEL
LIN {X 0,Y 373.319,Z 559.514,A -85,B 0,C 180,E1 17292.216,E2 17292.216} C_VEL
LIN {X 0,Y 369.655,Z 557.269,A -85,B 0,C 180,E1 17288.869,E2 17288.869} C_VEL
LIN {X 0,Y 367.687,Z 553.582,A -85,B 0,C 180,E1 17285.853,E2 17285.853} C_VEL
LIN {X 0,Y 367.455,Z 552.808,A -85,B 0,C 180,E1 17285.309,E2 17285.309} C_VEL
LIN {X 0,Y 366.515,Z 552.591,A -85,B 0,C 180,E1 17277.342,E2 17277.342} C_VEL
LIN {X 0,Y 367.573,Z 553.015,A -85,B 0,C 180,E1 17274.929,E2 17274.929} C_VEL
LIN {X 0,Y 369.041,Z 556.511,A -85,B 0,C 180,E1 17272.371,E2 17272.371} C_VEL
LIN {X 0,Y 372.562,Z 559.201,A -85,B 0,C 180,E1 17268.859,E2 17268.859} C_VEL
LIN {X 0,Y 373.455,Z 559.809,A -85,B 0,C 180,E1 17268.143,E2 17268.143} C_VEL
LIN {X 0,Y 375.532,Z 563.51,A -85,B 0,C 180,E1 17266.45,E2 17266.45} C_VEL
LIN {X 0,Y 379.057,Z 566.307,A -85,B 0,C 180,E1 17264.236,E2 17264.236} C_VEL
LIN {X 0,Y 381.765,Z 570.328,A -85,B 0,C 180,E1 17262.629,E2 17262.629} C_VEL
LIN {X 0,Y 384.462,Z 572.77,A -85,B 0,C 180,E1 17261.266,E2 17261.266} C_VEL
LIN {X 0,Y 387.527,Z 576.9,A -85,B 0,C 180,E1 17259.774,E2 17259.774} C_VEL
LIN {X 0,Y 389.531,Z 578.86,A -85,B 0,C 180,E1 17258.9,E2 17258.9} C_VEL
LIN {X 0,Y 393.068,Z 583.293,A -85,B 0,C 180,E1 17257.412,E2 17257.412} C_VEL
LIN {X 0,Y 394.96,Z 585.727,A -85,B 0,C 180,E1 17256.66,E2 17256.66} C_VEL
LIN {X 0,Y 400.966,Z 593.657,A -85,B 0,C 180,E1 17254.444,E2 17254.444} C_VEL
LIN {X 0,Y 409.462,Z 605.825,A -85,B 0,C 180,E1 17251.645,E2 17251.645} C_VEL
LIN {X 0,Y 419.361,Z 620.99,A -85,B 0,C 180,E1 17248.764,E2 17248.764} C_VEL
LIN {X 0,Y 427.135,Z 634.041,A -85,B 0,C 180,E1 17246.709,E2 17246.709} C_VEL
LIN {X 0,Y 416.369,Z 847.823,A -85,B 0,C 180,E1 17242.622,E2 17242.622} C_VEL
LIN {X 0,Y 414.03,Z 890.394,A -85,B 0,C 180,E1 17241.777,E2 17241.777} C_VEL
LIN {X 0,Y 411.543,Z 913.012,A -85,B 0,C 180,E1 17241.152,E2 17241.152} C_VEL
LIN {X 0,Y 408.427,Z 934.86,A -85,B 0,C 180,E1 17240.346,E2 17240.346} C_VEL
LIN {X 0,Y 404.681,Z 955.903,A -85,B 0,C 180,E1 17239.333,E2 17239.333} C_VEL
LIN {X 0,Y 400.237,Z 977.511,A -85,B 0,C 180,E1 17238.044,E2 17238.044} C_VEL
LIN {X 0,Y 395.62,Z 997.163,A -85,B 0,C 180,E1 17236.602,E2 17236.602} C_VEL
LIN {X 0,Y 390.105,Z 1018.543,A -85,B 0,C 180,E1 17234.713,E2 17234.713} C_VEL
LIN {X 0,Y 385.022,Z 1036.851,A -85,B 0,C 180,E1 17232.778,E2 17232.778} C_VEL
LIN {X 0,Y 379.421,Z 1055.829,A -85,B 0,C 180,E1 17230.397,E2 17230.397} C_VEL
LIN {X 0,Y 374.206,Z 1073.125,A -85,B 0,C 180,E1 17227.85,E2 17227.85} C_VEL
LIN {X 0,Y 369.267,Z 1089.182,A -85,B 0,C 180,E1 17225.032,E2 17225.032} C_VEL
LIN {X 0,Y 364.745,Z 1104.265,A -85,B 0,C 180,E1 17221.942,E2 17221.942} C_VEL
LIN {X 0,Y 361.215,Z 1116.575,A -85,B 0,C 180,E1 17218.973,E2 17218.973} C_VEL
LIN {X 0,Y 357.824,Z 1129.464,A -85,B 0,C 180,E1 17215.31,E2 17215.31} C_VEL
LIN {X 0,Y 355.476,Z 1139.688,A -85,B 0,C 180,E1 17211.845,E2 17211.845} C_VEL
LIN {X 0,Y 353.794,Z 1148.326,A -85,B 0,C 180,E1 17208.275,E2 17208.275} C_VEL
LIN {X 0,Y 352.764,Z 1155.276,A -85,B 0,C 180,E1 17204.779,E2 17204.779} C_VEL
LIN {X 0,Y 352.209,Z 1160.819,A -85,B 0,C 180,E1 17201.13,E2 17201.13} C_VEL
LIN {X 0,Y 351.987,Z 1164.531,A -85,B 0,C 180,E1 17197.836,E2 17197.836} C_VEL
LIN {X 0,Y 351.937,Z 1167.094,A -85,B 0,C 180,E1 17194.236,E2 17194.236} C_VEL
LIN {X 0,Y 351.93,Z 1168.06,A -85,B 0,C 180,E1 17191.139,E2 17191.139} C_VEL
LIN {X 0,Y 351.938,Z 1167.918,A -85,B 0,C 180,E1 17187.883,E2 17187.883} C_VEL
LIN {X 0,Y 351.931,Z 1166.216,A -85,B 0,C 180,E1 17184.293,E2 17184.293} C_VEL
LIN {X 0,Y 352.049,Z 1163.376,A -85,B 0,C 180,E1 17181.013,E2 17181.013} C_VEL
LIN {X 0,Y 352.403,Z 1158.494,A -85,B 0,C 180,E1 17177.214,E2 17177.214} C_VEL
LIN {X 0,Y 353.102,Z 1152.78,A -85,B 0,C 180,E1 17173.888,E2 17173.888} C_VEL
LIN {X 0,Y 354.51,Z 1144.463,A -85,B 0,C 180,E1 17170.045,E2 17170.045} C_VEL
LIN {X 0,Y 356.377,Z 1135.594,A -85,B 0,C 180,E1 17166.697,E2 17166.697} C_VEL
LIN {X 0,Y 359.095,Z 1124.462,A -85,B 0,C 180,E1 17163.187,E2 17163.187} C_VEL
LIN {X 0,Y 362.512,Z 1112.029,A -85,B 0,C 180,E1 17159.868,E2 17159.868} C_VEL
LIN {X 0,Y 366.553,Z 1098.146,A -85,B 0,C 180,E1 17156.751,E2 17156.751} C_VEL
LIN {X 0,Y 371.29,Z 1082.592,A -85,B 0,C 180,E1 17153.753,E2 17153.753} C_VEL
LIN {X 0,Y 376.167,Z 1066.568,A -85,B 0,C 180,E1 17151.149,E2 17151.149} C_VEL
LIN {X 0,Y 381.693,Z 1048.144,A -85,B 0,C 180,E1 17148.59,E2 17148.59} C_VEL
LIN {X 0,Y 386.859,Z 1030.252,A -85,B 0,C 180,E1 17146.492,E2 17146.492} C_VEL
LIN {X 0,Y 392.393,Z 1009.841,A -85,B 0,C 180,E1 17144.481,E2 17144.481} C_VEL
LIN {X 0,Y 397.196,Z 990.724,A -85,B 0,C 180,E1 17142.9,E2 17142.9} C_VEL
LIN {X 0,Y 401.927,Z 969.476,A -85,B 0,C 180,E1 17141.453,E2 17141.453} C_VEL
LIN {X 0,Y 405.913,Z 949.306,A -85,B 0,C 180,E1 17140.325,E2 17140.325} C_VEL
LIN {X 0,Y 409.608,Z 926.654,A -85,B 0,C 180,E1 17139.33,E2 17139.33} C_VEL
LIN {X 0,Y 412.565,Z 904.662,A -85,B 0,C 180,E1 17138.593,E2 17138.593} C_VEL
LIN {X 0,Y 414.62,Z 881.108,A -85,B 0,C 180,E1 17138.028,E2 17138.028} C_VEL
LIN {X 0,Y 424.436,Z 684.686,A -85,B 0,C 180,E1 17134.264,E2 17134.264} C_VEL
LIN {X 0,Y 426.979,Z 633.72,A -85,B 0,C 180,E1 17133.267,E2 17133.267} C_VEL
LIN {X 0,Y 417.946,Z 618.945,A -85,B 0,C 180,E1 17130.873,E2 17130.873} C_VEL
LIN {X 0,Y 409.279,Z 605.612,A -85,B 0,C 180,E1 17128.329,E2 17128.329} C_VEL
LIN {X 0,Y 402.287,Z 595.695,A -85,B 0,C 180,E1 17126.059,E2 17126.059} C_VEL
LIN {X 0,Y 397.183,Z 588.494,A -85,B 0,C 180,E1 17124.225,E2 17124.225} C_VEL
LIN {X 0,Y 393.134,Z 583.36,A -85,B 0,C 180,E1 17122.663,E2 17122.663} C_VEL
LIN {X 0,Y 389.496,Z 578.838,A -85,B 0,C 180,E1 17121.141,E2 17121.141} C_VEL
LIN {X 0,Y 385.093,Z 573.896,A -85,B 0,C 180,E1 17119.135,E2 17119.135} C_VEL
LIN {X 0,Y 383.913,Z 572.075,A -85,B 0,C 180,E1 17118.526,E2 17118.526} C_VEL
LIN {X 0,Y 380.456,Z 568.764,A -85,B 0,C 180,E1 17116.724,E2 17116.724} C_VEL
LIN {X 0,Y 378.672,Z 565.874,A -85,B 0,C 180,E1 17115.624,E2 17115.624} C_VEL
LIN {X 0,Y 375.379,Z 563.342,A -85,B 0,C 180,E1 17113.556,E2 17113.556} C_VEL
LIN {X 0,Y 373.351,Z 559.595,A -85,B 0,C 180,E1 17111.9,E2 17111.9} C_VEL
LIN {X 0,Y 369.231,Z 556.746,A -85,B 0,C 180,E1 17108.095,E2 17108.095} C_VEL
LIN {X 0,Y 367.645,Z 553.438,A -85,B 0,C 180,E1 17105.618,E2 17105.618} C_VEL
LIN {X 0,Y 367.426,Z 552.802,A -85,B 0,C 180,E1 17105.152,E2 17105.152} C_VEL
LIN {X 0,Y 366.127,Z 552.479,A -85,B 0,C 180,E1 17097.339,E2 17097.339} C_VEL
LIN {X 0,Y 367.532,Z 553.001,A -85,B 0,C 180,E1 17094.066,E2 17094.066} C_VEL
LIN {X 0,Y 369.026,Z 556.486,A -85,B 0,C 180,E1 17091.587,E2 17091.587} C_VEL
LIN {X 0,Y 372.642,Z 559.239,A -85,B 0,C 180,E1 17088.076,E2 17088.076} C_VEL
LIN {X 0,Y 373.449,Z 559.848,A -85,B 0,C 180,E1 17087.435,E2 17087.435} C_VEL
LIN {X 0,Y 375.454,Z 563.443,A -85,B 0,C 180,E1 17085.818,E2 17085.818} C_VEL
LIN {X 0,Y 379.063,Z 566.342,A -85,B 0,C 180,E1 17083.567,E2 17083.567} C_VEL
LIN {X 0,Y 381.725,Z 570.336,A -85,B 0,C 180,E1 17081.996,E2 17081.996} C_VEL
LIN {X 0,Y 384.368,Z 572.687,A -85,B 0,C 180,E1 17080.669,E2 17080.669} C_VEL
LIN {X 0,Y 387.527,Z 576.881,A -85,B 0,C 180,E1 17079.142,E2 17079.142} C_VEL
LIN {X 0,Y 389.538,Z 578.887,A -85,B 0,C 180,E1 17078.268,E2 17078.268} C_VEL
LIN {X 0,Y 393.27,Z 583.495,A -85,B 0,C 180,E1 17076.712,E2 17076.712} C_VEL
LIN {X 0,Y 399.366,Z 591.186,A -85,B 0,C 180,E1 17074.413,E2 17074.413} C_VEL
LIN {X 0,Y 403.987,Z 597.151,A -85,B 0,C 180,E1 17072.83,E2 17072.83} C_VEL
LIN {X 0,Y 410.959,Z 606.425,A -85,B 0,C 180,E1 17070.643,E2 17070.643} C_VEL
LIN {X 0,Y 420.098,Z 619.199,A -85,B 0,C 180,E1 17068.064,E2 17068.064} C_VEL
LIN {X 0,Y 426.991,Z 629.658,A -85,B 0,C 180,E1 17066.28,E2 17066.28} C_VEL
LIN {X 0,Y 416.478,Z 836.553,A -85,B 0,C 180,E1 17062.33,E2 17062.33} C_VEL
LIN {X 0,Y 414.398,Z 872.225,A -85,B 0,C 180,E1 17061.609,E2 17061.609} C_VEL
LIN {X 0,Y 412.055,Z 894.347,A -85,B 0,C 180,E1 17060.968,E2 17060.968} C_VEL
LIN {X 0,Y 408.723,Z 918.172,A -85,B 0,C 180,E1 17060.024,E2 17060.024} C_VEL
LIN {X 0,Y 405.274,Z 937.951,A -85,B 0,C 180,E1 17059.021,E2 17059.021} C_VEL
LIN {X 0,Y 400.812,Z 959.614,A -85,B 0,C 180,E1 17057.659,E2 17057.659} C_VEL
LIN {X 0,Y 396.497,Z 978.022,A -85,B 0,C 180,E1 17056.26,E2 17056.26} C_VEL
LIN {X 0,Y 391.075,Z 998.745,A -85,B 0,C 180,E1 17054.368,E2 17054.368} C_VEL
LIN {X 0,Y 385.835,Z 1017.251,A -85,B 0,C 180,E1 17052.359,E2 17052.359} C_VEL
LIN {X 0,Y 380.473,Z 1034.823,A -85,B 0,C 180,E1 17050.08,E2 17050.08} C_VEL
LIN {X 0,Y 375.35,Z 1051.256,A -85,B 0,C 180,E1 17047.591,E2 17047.591} C_VEL
LIN {X 0,Y 370.216,Z 1067.06,A -85,B 0,C 180,E1 17044.741,E2 17044.741} C_VEL
LIN {X 0,Y 365.407,Z 1082.195,A -85,B 0,C 180,E1 17041.51,E2 17041.51} C_VEL
LIN {X 0,Y 361.623,Z 1094.538,A -85,B 0,C 180,E1 17038.397,E2 17038.397} C_VEL
LIN {X 0,Y 358.29,Z 1106.048,A -85,B 0,C 180,E1 17034.923,E2 17034.923} C_VEL
LIN {X 0,Y 355.821,Z 1115.8,A -85,B 0,C 180,E1 17031.427,E2 17031.427} C_VEL
LIN {X 0,Y 354.967,Z 1119.504,A -85,B 0,C 180,E1 17029.86,E2 17029.86} C_VEL
LIN {X 0,Y 353.418,Z 1122.284,A -85,B 0,C 180,E1 17028.713,E2 17028.713} C_VEL
LIN {X 0,Y 346.065,Z 1129.048,A -85,B 0,C 180,E1 17025.634,E2 17025.634} C_VEL
LIN {X 0,Y 345.026,Z 1130.769,A -85,B 0,C 180,E1 17024.577,E2 17024.577} C_VEL
LIN {X 0,Y 344.371,Z 1135.544,A -85,B 0,C 180,E1 17021.048,E2 17021.048} C_VEL
LIN {X 0,Y 344.038,Z 1139.236,A -85,B 0,C 180,E1 17017.347,E2 17017.347} C_VEL
LIN {X 0,Y 343.953,Z 1141.249,A -85,B 0,C 180,E1 17013.834,E2 17013.834} C_VEL
LIN {X 0,Y 343.929,Z 1142.031,A -85,B 0,C 180,E1 17010.667,E2 17010.667} C_VEL
LIN {X 0,Y 343.937,Z 1141.615,A -85,B 0,C 180,E1 17007.001,E2 17007.001} C_VEL
LIN {X 0,Y 344.004,Z 1139.953,A -85,B 0,C 180,E1 17003.659,E2 17003.659} C_VEL
LIN {X 0,Y 344.237,Z 1136.836,A -85,B 0,C 180,E1 16999.948,E2 16999.948} C_VEL
LIN {X 0,Y 344.804,Z 1132.135,A -85,B 0,C 180,E1 16996.272,E2 16996.272} C_VEL
LIN {X 0,Y 345.921,Z 1125.904,A -85,B 0,C 180,E1 16992.506,E2 16992.506} C_VEL
LIN {X 0,Y 347.599,Z 1118.29,A -85,B 0,C 180,E1 16988.927,E2 16988.927} C_VEL
LIN {X 0,Y 350.182,Z 1108.629,A -85,B 0,C 180,E1 16985.183,E2 16985.183} C_VEL
LIN {X 0,Y 353.347,Z 1098.042,A -85,B 0,C 180,E1 16981.8,E2 16981.8} C_VEL
LIN {X 0,Y 357.578,Z 1084.919,A -85,B 0,C 180,E1 16978.286,E2 16978.286} C_VEL
LIN {X 0,Y 361.993,Z 1071.832,A -85,B 0,C 180,E1 16975.32,E2 16975.32} C_VEL
LIN {X 0,Y 367.127,Z 1056.578,A -85,B 0,C 180,E1 16972.407,E2 16972.407} C_VEL
LIN {X 0,Y 372.529,Z 1040.594,A -85,B 0,C 180,E1 16969.797,E2 16969.797} C_VEL
LIN {X 0,Y 378.114,Z 1023.028,A -85,B 0,C 180,E1 16967.394,E2 16967.394} C_VEL
LIN {X 0,Y 383.87,Z 1004.121,A -85,B 0,C 180,E1 16965.206,E2 16965.206} C_VEL
LIN {X 0,Y 388.971,Z 985.864,A -85,B 0,C 180,E1 16963.434,E2 16963.434} C_VEL
LIN {X 0,Y 394.397,Z 964.443,A -85,B 0,C 180,E1 16961.703,E2 16961.703} C_VEL
LIN {X 0,Y 398.405,Z 946.486,A -85,B 0,C 180,E1 16960.498,E2 16960.498} C_VEL
LIN {X 0,Y 402.667,Z 924.385,A -85,B 0,C 180,E1 16959.286,E2 16959.286} C_VEL
LIN {X 0,Y 405.738,Z 904.981,A -85,B 0,C 180,E1 16958.44,E2 16958.44} C_VEL
LIN {X 0,Y 408.638,Z 881.704,A -85,B 0,C 180,E1 16957.663,E2 16957.663} C_VEL
LIN {X 0,Y 410.44,Z 860.136,A -85,B 0,C 180,E1 16957.147,E2 16957.147} C_VEL
LIN {X 0,Y 421.067,Z 658.724,A -85,B 0,C 180,E1 16953.271,E2 16953.271} C_VEL
LIN {X 0,Y 422.418,Z 633.75,A -85,B 0,C 180,E1 16952.787,E2 16952.787} C_VEL
LIN {X 0,Y 412.762,Z 619.52,A -85,B 0,C 180,E1 16950.139,E2 16950.139} C_VEL
LIN {X 0,Y 403.428,Z 606.524,A -85,B 0,C 180,E1 16947.251,E2 16947.251} C_VEL
LIN {X 0,Y 395.764,Z 596.499,A -85,B 0,C 180,E1 16944.557,E2 16944.557} C_VEL
LIN {X 0,Y 390.89,Z 590.482,A -85,B 0,C 180,E1 16942.642,E2 16942.642} C_VEL
LIN {X 0,Y 386.723,Z 585.256,A -85,B 0,C 180,E1 16940.824,E2 16940.824} C_VEL
LIN {X 0,Y 383.222,Z 581.195,A -85,B 0,C 180,E1 16939.153,E2 16939.153} C_VEL
LIN {X 0,Y 382.198,Z 579.694,A -85,B 0,C 180,E1 16938.613,E2 16938.613} C_VEL
LIN {X 0,Y 378.844,Z 576.291,A -85,B 0,C 180,E1 16936.798,E2 16936.798} C_VEL
LIN {X 0,Y 377.1,Z 573.548,A -85,B 0,C 180,E1 16935.691,E2 16935.691} C_VEL
LIN {X 0,Y 373.828,Z 570.798,A -85,B 0,C 180,E1 16933.535,E2 16933.535} C_VEL
LIN {X 0,Y 371.969,Z 567.341,A -85,B 0,C 180,E1 16931.946,E2 16931.946} C_VEL
LIN {X 0,Y 368.421,Z 565.006,A -85,B 0,C 180,E1 16928.585,E2 16928.585} C_VEL
LIN {X 0,Y 366.557,Z 561.271,A -85,B 0,C 180,E1 16925.557,E2 16925.557} C_VEL
LIN {X 0,Y 366.316,Z 560.721,A -85,B 0,C 180,E1 16925.011,E2 16925.011} C_VEL
LIN {X 0,Y 365.591,Z 560.547,A -85,B 0,C 180,E1 16917.179,E2 16917.179} C_VEL
LIN {X 0,Y 366.506,Z 560.99,A -85,B 0,C 180,E1 16915.071,E2 16915.071} C_VEL
LIN {X 0,Y 368.062,Z 564.55,A -85,B 0,C 180,E1 16912.351,E2 16912.351} C_VEL
LIN {X 0,Y 371.794,Z 567.233,A -85,B 0,C 180,E1 16908.679,E2 16908.679} C_VEL
LIN {X 0,Y 374.665,Z 571.776,A -85,B 0,C 180,E1 16906.339,E2 16906.339} C_VEL
LIN {X 0,Y 377.584,Z 574.136,A -85,B 0,C 180,E1 16904.488,E2 16904.488} C_VEL
LIN {X 0,Y 380.396,Z 578.153,A -85,B 0,C 180,E1 16902.801,E2 16902.801} C_VEL
LIN {X 0,Y 382.768,Z 580.394,A -85,B 0,C 180,E1 16901.575,E2 16901.575} C_VEL
LIN {X 0,Y 386.1,Z 584.741,A -85,B 0,C 180,E1 16899.933,E2 16899.933} C_VEL
LIN {X 0,Y 387.752,Z 586.499,A -85,B 0,C 180,E1 16899.195,E2 16899.195} C_VEL
LIN {X 0,Y 391.566,Z 591.123,A -85,B 0,C 180,E1 16897.572,E2 16897.572} C_VEL
LIN {X 0,Y 398.658,Z 600.828,A -85,B 0,C 180,E1 16894.842,E2 16894.842} C_VEL
LIN {X 0,Y 407.124,Z 613.138,A -85,B 0,C 180,E1 16891.986,E2 16891.986} C_VEL
LIN {X 0,Y 417.328,Z 629.188,A -85,B 0,C 180,E1 16888.956,E2 16888.956} C_VEL
LIN {X 0,Y 422.523,Z 638.267,A -85,B 0,C 180,E1 16887.534,E2 16887.534} C_VEL
LIN {X 0,Y 411.343,Z 851.326,A -85,B 0,C 180,E1 16883.44,E2 16883.44} C_VEL
LIN {X 0,Y 409.05,Z 890.585,A -85,B 0,C 180,E1 16882.651,E2 16882.651} C_VEL
LIN {X 0,Y 406.511,Z 912.917,A -85,B 0,C 180,E1 16882.031,E2 16882.031} C_VEL
LIN {X 0,Y 403.177,Z 935.308,A -85,B 0,C 180,E1 16881.199,E2 16881.199} C_VEL
LIN {X 0,Y 399.434,Z 955.606,A -85,B 0,C 180,E1 16880.217,E2 16880.217} C_VEL
LIN {X 0,Y 394.735,Z 977.576,A -85,B 0,C 180,E1 16878.9,E2 16878.9} C_VEL
LIN {X 0,Y 389.97,Z 997.087,A -85,B 0,C 180,E1 16877.46,E2 16877.46} C_VEL
LIN {X 0,Y 384.062,Z 1018.979,A -85,B 0,C 180,E1 16875.506,E2 16875.506} C_VEL
LIN {X 0,Y 378.571,Z 1037.932,A -85,B 0,C 180,E1 16873.473,E2 16873.473} C_VEL
LIN {X 0,Y 373.137,Z 1055.443,A -85,B 0,C 180,E1 16871.237,E2 16871.237} C_VEL
LIN {X 0,Y 367.745,Z 1072.457,A -85,B 0,C 180,E1 16868.707,E2 16868.707} C_VEL
LIN {X 0,Y 362.698,Z 1088.01,A -85,B 0,C 180,E1 16865.957,E2 16865.957} C_VEL
LIN {X 0,Y 358.117,Z 1102.524,A -85,B 0,C 180,E1 16862.986,E2 16862.986} C_VEL
LIN {X 0,Y 354.088,Z 1115.614,A -85,B 0,C 180,E1 16859.8,E2 16859.8} C_VEL
LIN {X 0,Y 350.569,Z 1128.097,A -85,B 0,C 180,E1 16856.236,E2 16856.236} C_VEL
LIN {X 0,Y 348.046,Z 1138.105,A -85,B 0,C 180,E1 16852.819,E2 16852.819} C_VEL
LIN {X 0,Y 346.031,Z 1147.639,A -85,B 0,C 180,E1 16848.882,E2 16848.882} C_VEL
LIN {X 0,Y 344.927,Z 1154.346,A -85,B 0,C 180,E1 16845.467,E2 16845.467} C_VEL
LIN {X 0,Y 344.248,Z 1160.301,A -85,B 0,C 180,E1 16841.561,E2 16841.561} C_VEL
LIN {X 0,Y 344.013,Z 1164.065,A -85,B 0,C 180,E1 16838.187,E2 16838.187} C_VEL
LIN {X 0,Y 343.938,Z 1166.723,A -85,B 0,C 180,E1 16834.502,E2 16834.502} C_VEL
LIN {X 0,Y 343.94,Z 1167.737,A -85,B 0,C 180,E1 16831.332,E2 16831.332} C_VEL
LIN {X 0,Y 343.942,Z 1167.666,A -85,B 0,C 180,E1 16828.167,E2 16828.167} C_VEL
LIN {X 0,Y 343.934,Z 1166.149,A -85,B 0,C 180,E1 16824.494,E2 16824.494} C_VEL
LIN {X 0,Y 344.042,Z 1163.403,A -85,B 0,C 180,E1 16821.139,E2 16821.139} C_VEL
LIN {X 0,Y 344.376,Z 1158.973,A -85,B 0,C 180,E1 16817.422,E2 16817.422} C_VEL
LIN {X 0,Y 345.108,Z 1153.095,A -85,B 0,C 180,E1 16813.851,E2 16813.851} C_VEL
LIN {X 0,Y 346.487,Z 1145.398,A -85,B 0,C 180,E1 16810.091,E2 16810.091} C_VEL
LIN {X 0,Y 348.497,Z 1136.221,A -85,B 0,C 180,E1 16806.496,E2 16806.496} C_VEL
LIN {X 0,Y 351.481,Z 1124.732,A -85,B 0,C 180,E1 16802.741,E2 16802.741} C_VEL
LIN {X 0,Y 354.869,Z 1113.01,A -85,B 0,C 180,E1 16799.525,E2 16799.525} C_VEL
LIN {X 0,Y 359.312,Z 1098.613,A -85,B 0,C 180,E1 16796.182,E2 16796.182} C_VEL
LIN {X 0,Y 364.112,Z 1083.686,A -85,B 0,C 180,E1 16793.227,E2 16793.227} C_VEL
LIN {X 0,Y 369.388,Z 1067.201,A -85,B 0,C 180,E1 16790.482,E2 16790.482} C_VEL
LIN {X 0,Y 374.942,Z 1049.677,A -85,B 0,C 180,E1 16787.983,E2 16787.983} C_VEL
LIN {X 0,Y 380.332,Z 1031.787,A -85,B 0,C 180,E1 16785.839,E2 16785.839} C_VEL
LIN {X 0,Y 386.227,Z 1011.166,A -85,B 0,C 180,E1 16783.757,E2 16783.757} C_VEL
LIN {X 0,Y 390.952,Z 993.135,A -85,B 0,C 180,E1 16782.234,E2 16782.234} C_VEL
LIN {X 0,Y 396.192,Z 970.944,A -85,B 0,C 180,E1 16780.679,E2 16780.679} C_VEL
LIN {X 0,Y 400.184,Z 951.602,A -85,B 0,C 180,E1 16779.577,E2 16779.577} C_VEL
LIN {X 0,Y 404.269,Z 928.108,A -85,B 0,C 180,E1 16778.513,E2 16778.513} C_VEL
LIN {X 0,Y 407.157,Z 907.622,A -85,B 0,C 180,E1 16777.809,E2 16777.809} C_VEL
LIN {X 0,Y 409.543,Z 883.258,A -85,B 0,C 180,E1 16777.194,E2 16777.194} C_VEL
LIN {X 0,Y 419.526,Z 692.202,A -85,B 0,C 180,E1 16773.506,E2 16773.506} C_VEL
LIN {X 0,Y 422.392,Z 637.778,A -85,B 0,C 180,E1 16772.442,E2 16772.442} C_VEL
LIN {X 0,Y 413.963,Z 623.95,A -85,B 0,C 180,E1 16770.118,E2 16770.118} C_VEL
LIN {X 0,Y 405.225,Z 610.349,A -85,B 0,C 180,E1 16767.438,E2 16767.438} C_VEL
LIN {X 0,Y 397.089,Z 598.684,A -85,B 0,C 180,E1 16764.628,E2 16764.628} C_VEL
LIN {X 0,Y 391.136,Z 590.738,A -85,B 0,C 180,E1 16762.309,E2 16762.309} C_VEL
LIN {X 0,Y 387.411,Z 585.978,A -85,B 0,C 180,E1 16760.706,E2 16760.706} C_VEL
LIN {X 0,Y 383.388,Z 581.478,A -85,B 0,C 180,E1 16758.828,E2 16758.828} C_VEL
LIN {X 0,Y 382.08,Z 579.583,A -85,B 0,C 180,E1 16758.144,E2 16758.144} C_VEL
LIN {X 0,Y 378.722,Z 576.13,A -85,B 0,C 180,E1 16756.33,E2 16756.33} C_VEL
LIN {X 0,Y 377.211,Z 573.63,A -85,B 0,C 180,E1 16755.37,E2 16755.37} C_VEL
LIN {X 0,Y 373.885,Z 570.901,A -85,B 0,C 180,E1 16753.217,E2 16753.217} C_VEL
LIN {X 0,Y 371.809,Z 567.241,A -85,B 0,C 180,E1 16751.478,E2 16751.478} C_VEL
LIN {X 0,Y 368.128,Z 564.627,A -85,B 0,C 180,E1 16747.962,E2 16747.962} C_VEL
LIN {X 0,Y 366.537,Z 561.264,A -85,B 0,C 180,E1 16745.4,E2 16745.4} C_VEL
LIN {X 0,Y 366.274,Z 560.714,A -85,B 0,C 180,E1 16744.854,E2 16744.854} C_VEL
LIN {X 0,Y 365.194,Z 560.436,A -85,B 0,C 180,E1 16737.175,E2 16737.175} C_VEL
LIN {X 0,Y 366.459,Z 560.996,A -85,B 0,C 180,E1 16734.206,E2 16734.206} C_VEL
LIN {X 0,Y 368.174,Z 564.686,A -85,B 0,C 180,E1 16731.41,E2 16731.41} C_VEL
LIN {X 0,Y 372.095,Z 567.637,A -85,B 0,C 180,E1 16727.704,E2 16727.704} C_VEL
LIN {X 0,Y 374.27,Z 571.375,A -85,B 0,C 180,E1 16725.93,E2 16725.93} C_VEL
LIN {X 0,Y 377.533,Z 574.064,A -85,B 0,C 180,E1 16723.854,E2 16723.854} C_VEL
LIN {X 0,Y 380.356,Z 578.166,A -85,B 0,C 180,E1 16722.166,E2 16722.166} C_VEL
LIN {X 0,Y 382.675,Z 580.314,A -85,B 0,C 180,E1 16720.977,E2 16720.977} C_VEL
LIN {X 0,Y 385.945,Z 584.576,A -85,B 0,C 180,E1 16719.37,E2 16719.37} C_VEL
LIN {X 0,Y 387.734,Z 586.49,A -85,B 0,C 180,E1 16718.572,E2 16718.572} C_VEL
LIN {X 0,Y 392.626,Z 592.687,A -85,B 0,C 180,E1 16716.513,E2 16716.513} C_VEL
LIN {X 0,Y 397.362,Z 598.72,A -85,B 0,C 180,E1 16714.714,E2 16714.714} C_VEL
LIN {X 0,Y 403.815,Z 607.067,A -85,B 0,C 180,E1 16712.498,E2 16712.498} C_VEL
LIN {X 0,Y 414.075,Z 621.384,A -85,B 0,C 180,E1 16709.369,E2 16709.369} C_VEL
LIN {X 0,Y 422.391,Z 633.787,A -85,B 0,C 180,E1 16707.109,E2 16707.109} C_VEL
LIN {X 0,Y 411.462,Z 840.345,A -85,B 0,C 180,E1 16703.145,E2 16703.145} C_VEL
LIN {X 0,Y 409.395,Z 873.352,A -85,B 0,C 180,E1 16702.466,E2 16702.466} C_VEL
LIN {X 0,Y 406.994,Z 895.181,A -85,B 0,C 180,E1 16701.827,E2 16701.827} C_VEL
LIN {X 0,Y 403.606,Z 918.484,A -85,B 0,C 180,E1 16700.898,E2 16700.898} C_VEL
LIN {X 0,Y 399.905,Z 938.964,A -85,B 0,C 180,E1 16699.853,E2 16699.853} C_VEL
LIN {X 0,Y 395.268,Z 960.52,A -85,B 0,C 180,E1 16698.483,E2 16698.483} C_VEL
LIN {X 0,Y 390.492,Z 980.117,A -85,B 0,C 180,E1 16696.973,E2 16696.973} C_VEL
LIN {X 0,Y 385.082,Z 999.782,A -85,B 0,C 180,E1 16695.141,E2 16695.141} C_VEL
LIN {X 0,Y 379.639,Z 1018.217,A -85,B 0,C 180,E1 16693.114,E2 16693.114} C_VEL
LIN {X 0,Y 374.168,Z 1035.303,A -85,B 0,C 180,E1 16690.866,E2 16690.866} C_VEL
LIN {X 0,Y 368.851,Z 1051.568,A -85,B 0,C 180,E1 16688.372,E2 16688.372} C_VEL
LIN {X 0,Y 363.743,Z 1066.542,A -85,B 0,C 180,E1 16685.645,E2 16685.645} C_VEL
LIN {X 0,Y 358.846,Z 1081.134,A -85,B 0,C 180,E1 16682.532,E2 16682.532} C_VEL
LIN {X 0,Y 354.85,Z 1093.258,A -85,B 0,C 180,E1 16679.463,E2 16679.463} C_VEL
LIN {X 0,Y 351.123,Z 1105.354,A -85,B 0,C 180,E1 16675.829,E2 16675.829} C_VEL
LIN {X 0,Y 348.503,Z 1114.794,A -85,B 0,C 180,E1 16672.432,E2 16672.432} C_VEL
LIN {X 0,Y 346.434,Z 1123.313,A -85,B 0,C 180,E1 16668.685,E2 16668.685} C_VEL
LIN {X 0,Y 345.162,Z 1129.909,A -85,B 0,C 180,E1 16665.113,E2 16665.113} C_VEL
LIN {X 0,Y 345.026,Z 1130.769,A -85,B 0,C 180,E1 16664.577,E2 16664.577} C_VEL
LIN {X 0,Y 343.752,Z 1132.666,A -85,B 0,C 180,E1 16663.341,E2 16663.341} C_VEL
LIN {X 0,Y 338.943,Z 1135.936,A -85,B 0,C 180,E1 16661.099,E2 16661.099} C_VEL
LIN {X 0,Y 336.426,Z 1137.794,A -85,B 0,C 180,E1 16659.475,E2 16659.475} C_VEL
LIN {X 0,Y 336.174,Z 1138.305,A -85,B 0,C 180,E1 16658.914,E2 16658.914} C_VEL
LIN {X 0,Y 335.989,Z 1141.073,A -85,B 0,C 180,E1 16655.122,E2 16655.122} C_VEL
LIN {X 0,Y 335.95,Z 1142.22,A -85,B 0,C 180,E1 16651.535,E2 16651.535} C_VEL
LIN {X 0,Y 335.951,Z 1142.211,A -85,B 0,C 180,E1 16648.295,E2 16648.295} C_VEL
LIN {X 0,Y 335.991,Z 1140.803,A -85,B 0,C 180,E1 16644.365,E2 16644.365} C_VEL
LIN {X 0,Y 336.181,Z 1138.225,A -85,B 0,C 180,E1 16640.905,E2 16640.905} C_VEL
LIN {X 0,Y 336.692,Z 1133.88,A -85,B 0,C 180,E1 16636.957,E2 16636.957} C_VEL
LIN {X 0,Y 337.66,Z 1128.312,A -85,B 0,C 180,E1 16633.308,E2 16633.308} C_VEL
LIN {X 0,Y 339.444,Z 1120.57,A -85,B 0,C 180,E1 16629.301,E2 16629.301} C_VEL
LIN {X 0,Y 341.726,Z 1112.202,A -85,B 0,C 180,E1 16625.819,E2 16625.819} C_VEL
LIN {X 0,Y 345.149,Z 1101.155,A -85,B 0,C 180,E1 16622.012,E2 16622.012} C_VEL
LIN {X 0,Y 348.959,Z 1089.877,A -85,B 0,C 180,E1 16618.761,E2 16618.761} C_VEL
LIN {X 0,Y 353.58,Z 1076.681,A -85,B 0,C 180,E1 16615.559,E2 16615.559} C_VEL
LIN {X 0,Y 358.743,Z 1062.278,A -85,B 0,C 180,E1 16612.585,E2 16612.585} C_VEL
LIN {X 0,Y 364.308,Z 1046.41,A -85,B 0,C 180,E1 16609.837,E2 16609.837} C_VEL
LIN {X 0,Y 370.197,Z 1029.338,A -85,B 0,C 180,E1 16607.319,E2 16607.319} C_VEL
LIN {X 0,Y 375.793,Z 1011.908,A -85,B 0,C 180,E1 16605.164,E2 16605.164} C_VEL
LIN {X 0,Y 381.61,Z 992.641,A -85,B 0,C 180,E1 16603.145,E2 16603.145} C_VEL
LIN {X 0,Y 386.659,Z 974.122,A -85,B 0,C 180,E1 16601.529,E2 16601.529} C_VEL
LIN {X 0,Y 391.963,Z 952.392,A -85,B 0,C 180,E1 16599.955,E2 16599.955} C_VEL
LIN {X 0,Y 396.221,Z 932.084,A -85,B 0,C 180,E1 16598.762,E2 16598.762} C_VEL
LIN {X 0,Y 400.206,Z 909.135,A -85,B 0,C 180,E1 16597.694,E2 16597.694} C_VEL
LIN {X 0,Y 403.143,Z 887.776,A -85,B 0,C 180,E1 16596.929,E2 16596.929} C_VEL
LIN {X 0,Y 405.373,Z 864.427,A -85,B 0,C 180,E1 16596.331,E2 16596.331} C_VEL
LIN {X 0,Y 415.98,Z 672.055,A -85,B 0,C 180,E1 16592.601,E2 16592.601} C_VEL
LIN {X 0,Y 417.844,Z 638,A -85,B 0,C 180,E1 16591.927,E2 16591.927} C_VEL
LIN {X 0,Y 407.828,Z 623.154,A -85,B 0,C 180,E1 16589.041,E2 16589.041} C_VEL
LIN {X 0,Y 399.222,Z 611.31,A -85,B 0,C 180,E1 16586.235,E2 16586.235} C_VEL
LIN {X 0,Y 393.351,Z 603.485,A -85,B 0,C 180,E1 16584.078,E2 16584.078} C_VEL
LIN {X 0,Y 388.919,Z 597.854,A -85,B 0,C 180,E1 16582.285,E2 16582.285} C_VEL
LIN {X 0,Y 384.825,Z 592.674,A -85,B 0,C 180,E1 16580.455,E2 16580.455} C_VEL
LIN {X 0,Y 381.271,Z 588.342,A -85,B 0,C 180,E1 16578.699,E2 16578.699} C_VEL
LIN {X 0,Y 380.106,Z 586.974,A -85,B 0,C 180,E1 16578.083,E2 16578.083} C_VEL
LIN {X 0,Y 376.899,Z 583.291,A -85,B 0,C 180,E1 16576.253,E2 16576.253} C_VEL
LIN {X 0,Y 375.656,Z 581.293,A -85,B 0,C 180,E1 16575.436,E2 16575.436} C_VEL
LIN {X 0,Y 372.454,Z 578.487,A -85,B 0,C 180,E1 16573.269,E2 16573.269} C_VEL
LIN {X 0,Y 370.628,Z 575.163,A -85,B 0,C 180,E1 16571.674,E2 16571.674} C_VEL
LIN {X 0,Y 367.076,Z 572.589,A -85,B 0,C 180,E1 16568.143,E2 16568.143} C_VEL
LIN {X 0,Y 365.41,Z 568.825,A -85,B 0,C 180,E1 16565.181,E2 16565.181} C_VEL
LIN {X 0,Y 364.32,Z 568.404,A -85,B 0,C 180,E1 16558.27,E2 16558.27} C_VEL
LIN {X 0,Y 365.444,Z 568.945,A -85,B 0,C 180,E1 16555.214,E2 16555.214} C_VEL
LIN {X 0,Y 367.085,Z 572.58,A -85,B 0,C 180,E1 16552.331,E2 16552.331} C_VEL
LIN {X 0,Y 370.804,Z 575.452,A -85,B 0,C 180,E1 16548.648,E2 16548.648} C_VEL
LIN {X 0,Y 373.167,Z 579.357,A -85,B 0,C 180,E1 16546.678,E2 16546.678} C_VEL
LIN {X 0,Y 376.123,Z 581.93,A -85,B 0,C 180,E1 16544.742,E2 16544.742} C_VEL
LIN {X 0,Y 379.164,Z 586.105,A -85,B 0,C 180,E1 16542.901,E2 16542.901} C_VEL
LIN {X 0,Y 381.087,Z 588.001,A -85,B 0,C 180,E1 16541.886,E2 16541.886} C_VEL
LIN {X 0,Y 384.522,Z 592.432,A -85,B 0,C 180,E1 16540.164,E2 16540.164} C_VEL
LIN {X 0,Y 386.135,Z 594.352,A -85,B 0,C 180,E1 16539.421,E2 16539.421} C_VEL
LIN {X 0,Y 390.675,Z 600.127,A -85,B 0,C 180,E1 16537.465,E2 16537.465} C_VEL
LIN {X 0,Y 396.46,Z 608.137,A -85,B 0,C 180,E1 16535.212,E2 16535.212} C_VEL
LIN {X 0,Y 404.597,Z 620.168,A -85,B 0,C 180,E1 16532.396,E2 16532.396} C_VEL
LIN {X 0,Y 414.313,Z 635.777,A -85,B 0,C 180,E1 16529.43,E2 16529.43} C_VEL
LIN {X 0,Y 418.006,Z 642.391,A -85,B 0,C 180,E1 16528.38,E2 16528.38} C_VEL
LIN {X 0,Y 406.388,Z 855.125,A -85,B 0,C 180,E1 16524.272,E2 16524.272} C_VEL
LIN {X 0,Y 404.154,Z 890.906,A -85,B 0,C 180,E1 16523.542,E2 16523.542} C_VEL
LIN {X 0,Y 401.568,Z 912.885,A -85,B 0,C 180,E1 16522.929,E2 16522.929} C_VEL
LIN {X 0,Y 398.018,Z 935.756,A -85,B 0,C 180,E1 16522.073,E2 16522.073} C_VEL
LIN {X 0,Y 394.284,Z 955.308,A -85,B 0,C 180,E1 16521.125,E2 16521.125} C_VEL
LIN {X 0,Y 389.419,Z 977.276,A -85,B 0,C 180,E1 16519.805,E2 16519.805} C_VEL
LIN {X 0,Y 384.531,Z 996.557,A -85,B 0,C 180,E1 16518.379,E2 16518.379} C_VEL
LIN {X 0,Y 378.654,Z 1017.561,A -85,B 0,C 180,E1 16516.51,E2 16516.51} C_VEL
LIN {X 0,Y 373.032,Z 1036.129,A -85,B 0,C 180,E1 16514.523,E2 16514.523} C_VEL
LIN {X 0,Y 367.19,Z 1054.292,A -85,B 0,C 180,E1 16512.213,E2 16512.213} C_VEL
LIN {X 0,Y 361.816,Z 1070.441,A -85,B 0,C 180,E1 16509.805,E2 16509.805} C_VEL
LIN {X 0,Y 356.227,Z 1086.838,A -85,B 0,C 180,E1 16506.917,E2 16506.917} C_VEL
LIN {X 0,Y 351.365,Z 1101.46,A -85,B 0,C 180,E1 16503.9,E2 16503.9} C_VEL
LIN {X 0,Y 347.035,Z 1114.653,A -85,B 0,C 180,E1 16500.661,E2 16500.661} C_VEL
LIN {X 0,Y 343.402,Z 1126.731,A -85,B 0,C 180,E1 16497.202,E2 16497.202} C_VEL
LIN {X 0,Y 340.5,Z 1137.324,A -85,B 0,C 180,E1 16493.538,E2 16493.538} C_VEL
LIN {X 0,Y 338.291,Z 1146.966,A -85,B 0,C 180,E1 16489.511,E2 16489.511} C_VEL
LIN {X 0,Y 337.067,Z 1153.727,A -85,B 0,C 180,E1 16486.014,E2 16486.014} C_VEL
LIN {X 0,Y 336.296,Z 1159.8,A -85,B 0,C 180,E1 16481.997,E2 16481.997} C_VEL
LIN {X 0,Y 336.028,Z 1163.597,A -85,B 0,C 180,E1 16478.556,E2 16478.556} C_VEL
LIN {X 0,Y 335.94,Z 1166.351,A -85,B 0,C 180,E1 16474.78,E2 16474.78} C_VEL
LIN {X 0,Y 335.947,Z 1167.437,A -85,B 0,C 180,E1 16471.364,E2 16471.364} C_VEL
LIN {X 0,Y 335.947,Z 1167.366,A -85,B 0,C 180,E1 16468.123,E2 16468.123} C_VEL
LIN {X 0,Y 335.936,Z 1165.848,A -85,B 0,C 180,E1 16464.363,E2 16464.363} C_VEL
LIN {X 0,Y 336.053,Z 1163.099,A -85,B 0,C 180,E1 16460.927,E2 16460.927} C_VEL
LIN {X 0,Y 336.413,Z 1158.666,A -85,B 0,C 180,E1 16457.12,E2 16457.12} C_VEL
LIN {X 0,Y 337.217,Z 1152.786,A -85,B 0,C 180,E1 16453.462,E2 16453.462} C_VEL
LIN {X 0,Y 338.698,Z 1145.086,A -85,B 0,C 180,E1 16449.613,E2 16449.613} C_VEL
LIN {X 0,Y 340.859,Z 1135.907,A -85,B 0,C 180,E1 16445.937,E2 16445.937} C_VEL
LIN {X 0,Y 344.11,Z 1124.218,A -85,B 0,C 180,E1 16442.043,E2 16442.043} C_VEL
LIN {X 0,Y 347.88,Z 1112.045,A -85,B 0,C 180,E1 16438.652,E2 16438.652} C_VEL
LIN {X 0,Y 352.473,Z 1097.957,A -85,B 0,C 180,E1 16435.349,E2 16435.349} C_VEL
LIN {X 0,Y 357.745,Z 1082.483,A -85,B 0,C 180,E1 16432.259,E2 16432.259} C_VEL
LIN {X 0,Y 363.292,Z 1065.935,A -85,B 0,C 180,E1 16429.494,E2 16429.494} C_VEL
LIN {X 0,Y 369.458,Z 1047.243,A -85,B 0,C 180,E1 16426.848,E2 16426.848} C_VEL
LIN {X 0,Y 375.096,Z 1029.401,A -85,B 0,C 180,E1 16424.726,E2 16424.726} C_VEL
LIN {X 0,Y 381.029,Z 1009.214,A -85,B 0,C 180,E1 16422.713,E2 16422.713} C_VEL
LIN {X 0,Y 386.232,Z 990.038,A -85,B 0,C 180,E1 16421.112,E2 16421.112} C_VEL
LIN {X 0,Y 391.34,Z 968.706,A -85,B 0,C 180,E1 16419.652,E2 16419.652} C_VEL
LIN {X 0,Y 395.855,Z 947.389,A -85,B 0,C 180,E1 16418.463,E2 16418.463} C_VEL
LIN {X 0,Y 399.766,Z 924.611,A -85,B 0,C 180,E1 16417.48,E2 16417.48} C_VEL
LIN {X 0,Y 403.01,Z 901.192,A -85,B 0,C 180,E1 16416.725,E2 16416.725} C_VEL
LIN {X 0,Y 405.029,Z 878.639,A -85,B 0,C 180,E1 16416.195,E2 16416.195} C_VEL
LIN {X 0,Y 415.96,Z 677.307,A -85,B 0,C 180,E1 16412.3,E2 16412.3} C_VEL
LIN {X 0,Y 417.88,Z 641.977,A -85,B 0,C 180,E1 16411.6,E2 16411.6} C_VEL
LIN {X 0,Y 409.741,Z 628.405,A -85,B 0,C 180,E1 16409.252,E2 16409.252} C_VEL
LIN {X 0,Y 401.544,Z 615.68,A -85,B 0,C 180,E1 16406.628,E2 16406.628} C_VEL
LIN {X 0,Y 394.112,Z 604.853,A -85,B 0,C 180,E1 16403.948,E2 16403.948} C_VEL
LIN {X 0,Y 388.984,Z 597.942,A -85,B 0,C 180,E1 16401.883,E2 16401.883} C_VEL
LIN {X 0,Y 384.709,Z 592.612,A -85,B 0,C 180,E1 16399.984,E2 16399.984} C_VEL
LIN {X 0,Y 381.157,Z 588.179,A -85,B 0,C 180,E1 16398.229,E2 16398.229} C_VEL
LIN {X 0,Y 379.985,Z 586.843,A -85,B 0,C 180,E1 16397.613,E2 16397.613} C_VEL
LIN {X 0,Y 376.655,Z 582.937,A -85,B 0,C 180,E1 16395.709,E2 16395.709} C_VEL
LIN {X 0,Y 375.509,Z 581.241,A -85,B 0,C 180,E1 16394.968,E2 16394.968} C_VEL
LIN {X 0,Y 372.212,Z 578.182,A -85,B 0,C 180,E1 16392.725,E2 16392.725} C_VEL
LIN {X 0,Y 370.465,Z 575.056,A -85,B 0,C 180,E1 16391.205,E2 16391.205} C_VEL
LIN {X 0,Y 366.907,Z 572.351,A -85,B 0,C 180,E1 16387.673,E2 16387.673} C_VEL
LIN {X 0,Y 365.374,Z 568.815,A -85,B 0,C 180,E1 16385.023,E2 16385.023} C_VEL
LIN {X 0,Y 364.013,Z 568.29,A -85,B 0,C 180,E1 16378.111,E2 16378.111} C_VEL
LIN {X 0,Y 365.36,Z 568.829,A -85,B 0,C 180,E1 16374.425,E2 16374.425} C_VEL
LIN {X 0,Y 367.073,Z 572.567,A -85,B 0,C 180,E1 16371.541,E2 16371.541} C_VEL
LIN {X 0,Y 370.791,Z 575.5,A -85,B 0,C 180,E1 16367.937,E2 16367.937} C_VEL
LIN {X 0,Y 373.089,Z 579.299,A -85,B 0,C 180,E1 16366.043,E2 16366.043} C_VEL
LIN {X 0,Y 376.069,Z 581.873,A -85,B 0,C 180,E1 16364.106,E2 16364.106} C_VEL
LIN {X 0,Y 378.991,Z 585.992,A -85,B 0,C 180,E1 16362.338,E2 16362.338} C_VEL
LIN {X 0,Y 381.06,Z 588.037,A -85,B 0,C 180,E1 16361.25,E2 16361.25} C_VEL
LIN {X 0,Y 384.524,Z 592.415,A -85,B 0,C 180,E1 16359.529,E2 16359.529} C_VEL
LIN {X 0,Y 386.065,Z 594.267,A -85,B 0,C 180,E1 16358.82,E2 16358.82} C_VEL
LIN {X 0,Y 390.537,Z 599.956,A -85,B 0,C 180,E1 16356.899,E2 16356.899} C_VEL
LIN {X 0,Y 395.28,Z 606.116,A -85,B 0,C 180,E1 16355.052,E2 16355.052} C_VEL
LIN {X 0,Y 401.441,Z 614.254,A -85,B 0,C 180,E1 16352.884,E2 16352.884} C_VEL
LIN {X 0,Y 411.229,Z 628.123,A -85,B 0,C 180,E1 16349.822,E2 16349.822} C_VEL
LIN {X 0,Y 417.854,Z 638.352,A -85,B 0,C 180,E1 16347.949,E2 16347.949} C_VEL
LIN {X 0,Y 406.555,Z 843.678,A -85,B 0,C 180,E1 16343.989,E2 16343.989} C_VEL
LIN {X 0,Y 404.437,Z 874.964,A -85,B 0,C 180,E1 16343.33,E2 16343.33} C_VEL
LIN {X 0,Y 401.964,Z 896.535,A -85,B 0,C 180,E1 16342.69,E2 16342.69} C_VEL
LIN {X 0,Y 398.457,Z 919.531,A -85,B 0,C 180,E1 16341.76,E2 16341.76} C_VEL
LIN {X 0,Y 394.554,Z 940.336,A -85,B 0,C 180,E1 16340.688,E2 16340.688} C_VEL
LIN {X 0,Y 389.885,Z 961.105,A -85,B 0,C 180,E1 16339.354,E2 16339.354} C_VEL
LIN {X 0,Y 384.772,Z 981.319,A -85,B 0,C 180,E1 16337.783,E2 16337.783} C_VEL
LIN {X 0,Y 379.377,Z 1000.093,A -85,B 0,C 180,E1 16336.014,E2 16336.014} C_VEL
LIN {X 0,Y 373.712,Z 1018.538,A -85,B 0,C 180,E1 16333.97,E2 16333.97} C_VEL
LIN {X 0,Y 367.793,Z 1036.214,A -85,B 0,C 180,E1 16331.617,E2 16331.617} C_VEL
LIN {X 0,Y 362.085,Z 1052.792,A -85,B 0,C 180,E1 16329.021,E2 16329.021} C_VEL
LIN {X 0,Y 356.771,Z 1067.686,A -85,B 0,C 180,E1 16326.252,E2 16326.252} C_VEL
LIN {X 0,Y 351.398,Z 1082.821,A -85,B 0,C 180,E1 16322.921,E2 16322.921} C_VEL
LIN {X 0,Y 347.149,Z 1095.164,A -85,B 0,C 180,E1 16319.696,E2 16319.696} C_VEL
LIN {X 0,Y 343.381,Z 1106.671,A -85,B 0,C 180,E1 16316.084,E2 16316.084} C_VEL
LIN {X 0,Y 340.547,Z 1116.42,A -85,B 0,C 180,E1 16312.439,E2 16312.439} C_VEL
LIN {X 0,Y 338.51,Z 1124.309,A -85,B 0,C 180,E1 16308.782,E2 16308.782} C_VEL
LIN {X 0,Y 337.146,Z 1131.038,A -85,B 0,C 180,E1 16304.953,E2 16304.953} C_VEL
LIN {X 0,Y 336.421,Z 1135.918,A -85,B 0,C 180,E1 16301.252,E2 16301.252} C_VEL
LIN {X 0,Y 336.174,Z 1138.305,A -85,B 0,C 180,E1 16298.914,E2 16298.914} C_VEL
LIN {X 0,Y 335.083,Z 1139.524,A -85,B 0,C 180,E1 16297.617,E2 16297.617} C_VEL
LIN {X 0,Y 328.588,Z 1141.834,A -85,B 0,C 180,E1 16294.031,E2 16294.031} C_VEL
LIN {X 0,Y 327.95,Z 1142.247,A -85,B 0,C 180,E1 16292.966,E2 16292.966} C_VEL
LIN {X 0,Y 327.939,Z 1142.62,A -85,B 0,C 180,E1 16289.127,E2 16289.127} C_VEL
LIN {X 0,Y 327.974,Z 1141.82,A -85,B 0,C 180,E1 16285.805,E2 16285.805} C_VEL
LIN {X 0,Y 328.111,Z 1139.633,A -85,B 0,C 180,E1 16281.942,E2 16281.942} C_VEL
LIN {X 0,Y 328.497,Z 1136.059,A -85,B 0,C 180,E1 16278.233,E2 16278.233} C_VEL
LIN {X 0,Y 329.356,Z 1130.97,A -85,B 0,C 180,E1 16274.325,E2 16274.325} C_VEL
LIN {X 0,Y 330.888,Z 1124.111,A -85,B 0,C 180,E1 16270.403,E2 16270.403} C_VEL
LIN {X 0,Y 333.259,Z 1115.644,A -85,B 0,C 180,E1 16266.483,E2 16266.483} C_VEL
LIN {X 0,Y 336.243,Z 1106.227,A -85,B 0,C 180,E1 16262.938,E2 16262.938} C_VEL
LIN {X 0,Y 340.535,Z 1093.918,A -85,B 0,C 180,E1 16259.081,E2 16259.081} C_VEL
LIN {X 0,Y 345.148,Z 1081.412,A -85,B 0,C 180,E1 16255.806,E2 16255.806} C_VEL
LIN {X 0,Y 350.324,Z 1067.573,A -85,B 0,C 180,E1 16252.766,E2 16252.766} C_VEL
LIN {X 0,Y 356.1,Z 1052.175,A -85,B 0,C 180,E1 16249.88,E2 16249.88} C_VEL
LIN {X 0,Y 362.205,Z 1035.184,A -85,B 0,C 180,E1 16247.229,E2 16247.229} C_VEL
LIN {X 0,Y 368.341,Z 1017.49,A -85,B 0,C 180,E1 16244.889,E2 16244.889} C_VEL
LIN {X 0,Y 374.047,Z 999.633,A -85,B 0,C 180,E1 16242.91,E2 16242.91} C_VEL
LIN {X 0,Y 379.893,Z 979.776,A -85,B 0,C 180,E1 16241.057,E2 16241.057} C_VEL
LIN {X 0,Y 385.052,Z 960.051,A -85,B 0,C 180,E1 16239.537,E2 16239.537} C_VEL
LIN {X 0,Y 390.176,Z 937.484,A -85,B 0,C 180,E1 16238.121,E2 16238.121} C_VEL
LIN {X 0,Y 394.282,Z 916.011,A -85,B 0,C 180,E1 16237.044,E2 16237.044} C_VEL
LIN {X 0,Y 397.674,Z 893.243,A -85,B 0,C 180,E1 16236.173,E2 16236.173} C_VEL
LIN {X 0,Y 400.297,Z 869.98,A -85,B 0,C 180,E1 16235.522,E2 16235.522} C_VEL
LIN {X 0,Y 404.767,Z 793.658,A -85,B 0,C 180,E1 16234.017,E2 16234.017} C_VEL
LIN {X 0,Y 413.404,Z 642.433,A -85,B 0,C 180,E1 16231.063,E2 16231.063} C_VEL
LIN {X 0,Y 404.76,Z 629.486,A -85,B 0,C 180,E1 16228.474,E2 16228.474} C_VEL
LIN {X 0,Y 395.351,Z 616.136,A -85,B 0,C 180,E1 16225.263,E2 16225.263} C_VEL
LIN {X 0,Y 390.185,Z 609.529,A -85,B 0,C 180,E1 16223.283,E2 16223.283} C_VEL
LIN {X 0,Y 386.8,Z 605.047,A -85,B 0,C 180,E1 16221.854,E2 16221.854} C_VEL
LIN {X 0,Y 382.945,Z 600.085,A -85,B 0,C 180,E1 16220.081,E2 16220.081} C_VEL
LIN {X 0,Y 379.344,Z 595.488,A -85,B 0,C 180,E1 16218.24,E2 16218.24} C_VEL
LIN {X 0,Y 375.258,Z 590.732,A -85,B 0,C 180,E1 16215.882,E2 16215.882} C_VEL
LIN {X 0,Y 374.219,Z 589.033,A -85,B 0,C 180,E1 16215.18,E2 16215.18} C_VEL
LIN {X 0,Y 370.994,Z 586.043,A -85,B 0,C 180,E1 16212.926,E2 16212.926} C_VEL
LIN {X 0,Y 369.296,Z 582.979,A -85,B 0,C 180,E1 16211.4,E2 16211.4} C_VEL
LIN {X 0,Y 365.867,Z 580.314,A -85,B 0,C 180,E1 16207.854,E2 16207.854} C_VEL
LIN {X 0,Y 364.216,Z 576.574,A -85,B 0,C 180,E1 16204.724,E2 16204.724} C_VEL
LIN {X 0,Y 363.752,Z 576.462,A -85,B 0,C 180,E1 16196.849,E2 16196.849} C_VEL
LIN {X 0,Y 364.386,Z 576.883,A -85,B 0,C 180,E1 16195.357,E2 16195.357} C_VEL
LIN {X 0,Y 366.109,Z 580.605,A -85,B 0,C 180,E1 16192.31,E2 16192.31} C_VEL
LIN {X 0,Y 369.475,Z 583.191,A -85,B 0,C 180,E1 16188.923,E2 16188.923} C_VEL
LIN {X 0,Y 371.885,Z 587.16,A -85,B 0,C 180,E1 16186.869,E2 16186.869} C_VEL
LIN {X 0,Y 374.618,Z 589.603,A -85,B 0,C 180,E1 16185.036,E2 16185.036} C_VEL
LIN {X 0,Y 377.802,Z 593.918,A -85,B 0,C 180,E1 16183.076,E2 16183.076} C_VEL
LIN {X 0,Y 379.484,Z 595.707,A -85,B 0,C 180,E1 16182.164,E2 16182.164} C_VEL
LIN {X 0,Y 383.104,Z 600.265,A -85,B 0,C 180,E1 16180.326,E2 16180.326} C_VEL
LIN {X 0,Y 388.602,Z 607.388,A -85,B 0,C 180,E1 16177.856,E2 16177.856} C_VEL
LIN {X 0,Y 394.28,Z 615.435,A -85,B 0,C 180,E1 16175.585,E2 16175.585} C_VEL
LIN {X 0,Y 402.087,Z 627.237,A -85,B 0,C 180,E1 16172.812,E2 16172.812} C_VEL
LIN {X 0,Y 411.326,Z 642.362,A -85,B 0,C 180,E1 16169.911,E2 16169.911} C_VEL
LIN {X 0,Y 413.581,Z 646.552,A -85,B 0,C 180,E1 16169.242,E2 16169.242} C_VEL
LIN {X 0,Y 401.499,Z 859.312,A -85,B 0,C 180,E1 16165.117,E2 16165.117} C_VEL
LIN {X 0,Y 399.294,Z 891.812,A -85,B 0,C 180,E1 16164.44,E2 16164.44} C_VEL
LIN {X 0,Y 396.664,Z 913.314,A -85,B 0,C 180,E1 16163.835,E2 16163.835} C_VEL
LIN {X 0,Y 392.924,Z 936.362,A -85,B 0,C 180,E1 16162.964,E2 16162.964} C_VEL
LIN {X 0,Y 388.967,Z 956.303,A -85,B 0,C 180,E1 16161.987,E2 16161.987} C_VEL
LIN {X 0,Y 383.674,Z 978.999,A -85,B 0,C 180,E1 16160.595,E2 16160.595} C_VEL
LIN {X 0,Y 378.58,Z 998.292,A -85,B 0,C 180,E1 16159.143,E2 16159.143} C_VEL
LIN {X 0,Y 372.42,Z 1019.184,A -85,B 0,C 180,E1 16157.235,E2 16157.235} C_VEL
LIN {X 0,Y 366.488,Z 1037.992,A -85,B 0,C 180,E1 16155.181,E2 16155.181} C_VEL
LIN {X 0,Y 360.38,Z 1055.949,A -85,B 0,C 180,E1 16152.823,E2 16152.823} C_VEL
LIN {X 0,Y 354.502,Z 1072.805,A -85,B 0,C 180,E1 16150.232,E2 16150.232} C_VEL
LIN {X 0,Y 348.947,Z 1088.245,A -85,B 0,C 180,E1 16147.406,E2 16147.406} C_VEL
LIN {X 0,Y 343.637,Z 1103.327,A -85,B 0,C 180,E1 16144.164,E2 16144.164} C_VEL
LIN {X 0,Y 339.341,Z 1115.856,A -85,B 0,C 180,E1 16140.973,E2 16140.973} C_VEL
LIN {X 0,Y 335.302,Z 1128.526,A -85,B 0,C 180,E1 16137.145,E2 16137.145} C_VEL
LIN {X 0,Y 332.427,Z 1138.729,A -85,B 0,C 180,E1 16133.458,E2 16133.458} C_VEL
LIN {X 0,Y 330.334,Z 1147.383,A -85,B 0,C 180,E1 16129.632,E2 16129.632} C_VEL
LIN {X 0,Y 328.977,Z 1154.667,A -85,B 0,C 180,E1 16125.694,E2 16125.694} C_VEL
LIN {X 0,Y 328.268,Z 1160.118,A -85,B 0,C 180,E1 16121.775,E2 16121.775} C_VEL
LIN {X 0,Y 328.007,Z 1163.954,A -85,B 0,C 180,E1 16118.06,E2 16118.06} C_VEL
LIN {X 0,Y 327.948,Z 1166.334,A -85,B 0,C 180,E1 16114.196,E2 16114.196} C_VEL
LIN {X 0,Y 327.943,Z 1167.184,A -85,B 0,C 180,E1 16111.048,E2 16111.048} C_VEL
LIN {X 0,Y 327.94,Z 1166.96,A -85,B 0,C 180,E1 16107.378,E2 16107.378} C_VEL
LIN {X 0,Y 327.959,Z 1165.166,A -85,B 0,C 180,E1 16103.656,E2 16103.656} C_VEL
LIN {X 0,Y 328.073,Z 1162.464,A -85,B 0,C 180,E1 16100.35,E2 16100.35} C_VEL
LIN {X 0,Y 328.516,Z 1157.835,A -85,B 0,C 180,E1 16096.446,E2 16096.446} C_VEL
LIN {X 0,Y 329.391,Z 1152.164,A -85,B 0,C 180,E1 16092.875,E2 16092.875} C_VEL
LIN {X 0,Y 331.101,Z 1143.942,A -85,B 0,C 180,E1 16088.753,E2 16088.753} C_VEL
LIN {X 0,Y 333.376,Z 1135.122,A -85,B 0,C 180,E1 16085.172,E2 16085.172} C_VEL
LIN {X 0,Y 336.845,Z 1123.514,A -85,B 0,C 180,E1 16081.257,E2 16081.257} C_VEL
LIN {X 0,Y 340.97,Z 1111.08,A -85,B 0,C 180,E1 16077.744,E2 16077.744} C_VEL
LIN {X 0,Y 345.752,Z 1097.194,A -85,B 0,C 180,E1 16074.46,E2 16074.46} C_VEL
LIN {X 0,Y 351.159,Z 1082.166,A -85,B 0,C 180,E1 16071.423,E2 16071.423} C_VEL
LIN {X 0,Y 356.974,Z 1065.618,A -85,B 0,C 180,E1 16068.622,E2 16068.622} C_VEL
LIN {X 0,Y 363.351,Z 1047.198,A -85,B 0,C 180,E1 16065.986,E2 16065.986} C_VEL
LIN {X 0,Y 369.08,Z 1029.808,A -85,B 0,C 180,E1 16063.894,E2 16063.894} C_VEL
LIN {X 0,Y 375.487,Z 1008.901,A -85,B 0,C 180,E1 16061.789,E2 16061.789} C_VEL
LIN {X 0,Y 380.872,Z 989.786,A -85,B 0,C 180,E1 16060.187,E2 16060.187} C_VEL
LIN {X 0,Y 386.005,Z 969.18,A -85,B 0,C 180,E1 16058.768,E2 16058.768} C_VEL
LIN {X 0,Y 390.58,Z 948.37,A -85,B 0,C 180,E1 16057.598,E2 16057.598} C_VEL
LIN {X 0,Y 394.707,Z 925.496,A -85,B 0,C 180,E1 16056.595,E2 16056.595} C_VEL
LIN {X 0,Y 398.074,Z 902.496,A -85,B 0,C 180,E1 16055.838,E2 16055.838} C_VEL
LIN {X 0,Y 400.257,Z 879.284,A -85,B 0,C 180,E1 16055.285,E2 16055.285} C_VEL
LIN {X 0,Y 411.521,Z 680.18,A -85,B 0,C 180,E1 16051.413,E2 16051.413} C_VEL
LIN {X 0,Y 413.416,Z 646.109,A -85,B 0,C 180,E1 16050.728,E2 16050.728} C_VEL
LIN {X 0,Y 405.803,Z 633.346,A -85,B 0,C 180,E1 16048.434,E2 16048.434} C_VEL
LIN {X 0,Y 398.704,Z 622.142,A -85,B 0,C 180,E1 16046.071,E2 16046.071} C_VEL
LIN {X 0,Y 391.711,Z 611.742,A -85,B 0,C 180,E1 16043.465,E2 16043.465} C_VEL
LIN {X 0,Y 386.855,Z 605.136,A -85,B 0,C 180,E1 16041.451,E2 16041.451} C_VEL
LIN {X 0,Y 382.824,Z 600.016,A -85,B 0,C 180,E1 16039.61,E2 16039.61} C_VEL
LIN {X 0,Y 379.225,Z 595.319,A -85,B 0,C 180,E1 16037.769,E2 16037.769} C_VEL
LIN {X 0,Y 375.193,Z 590.674,A -85,B 0,C 180,E1 16035.455,E2 16035.455} C_VEL
LIN {X 0,Y 374.07,Z 588.976,A -85,B 0,C 180,E1 16034.71,E2 16034.71} C_VEL
LIN {X 0,Y 370.845,Z 585.871,A -85,B 0,C 180,E1 16032.456,E2 16032.456} C_VEL
LIN {X 0,Y 369.131,Z 582.864,A -85,B 0,C 180,E1 16030.929,E2 16030.929} C_VEL
LIN {X 0,Y 365.582,Z 579.912,A -85,B 0,C 180,E1 16027.227,E2 16027.227} C_VEL
LIN {X 0,Y 364.16,Z 576.566,A -85,B 0,C 180,E1 16024.567,E2 16024.567} C_VEL
LIN {X 0,Y 363.29,Z 576.335,A -85,B 0,C 180,E1 16017.002,E2 16017.002} C_VEL
LIN {X 0,Y 364.297,Z 576.788,A -85,B 0,C 180,E1 16014.566,E2 16014.566} C_VEL
LIN {X 0,Y 366.098,Z 580.595,A -85,B 0,C 180,E1 16011.519,E2 16011.519} C_VEL
LIN {X 0,Y 369.457,Z 583.244,A -85,B 0,C 180,E1 16008.21,E2 16008.21} C_VEL
LIN {X 0,Y 371.807,Z 587.104,A -85,B 0,C 180,E1 16006.232,E2 16006.232} C_VEL
LIN {X 0,Y 374.561,Z 589.555,A -85,B 0,C 180,E1 16004.398,E2 16004.398} C_VEL
LIN {X 0,Y 377.63,Z 593.814,A -85,B 0,C 180,E1 16002.511,E2 16002.511} C_VEL
LIN {X 0,Y 379.391,Z 595.633,A -85,B 0,C 180,E1 16001.563,E2 16001.563} C_VEL
LIN {X 0,Y 383.107,Z 600.249,A -85,B 0,C 180,E1 15999.689,E2 15999.689} C_VEL
LIN {X 0,Y 388.628,Z 607.468,A -85,B 0,C 180,E1 15997.219,E2 15997.219} C_VEL
LIN {X 0,Y 393.391,Z 613.755,A -85,B 0,C 180,E1 15995.325,E2 15995.325} C_VEL
LIN {X 0,Y 399.276,Z 621.733,A -85,B 0,C 180,E1 15993.208,E2 15993.208} C_VEL
LIN {X 0,Y 408.409,Z 634.863,A -85,B 0,C 180,E1 15990.28,E2 15990.28} C_VEL
LIN {X 0,Y 413.412,Z 642.813,A -85,B 0,C 180,E1 15988.809,E2 15988.809} C_VEL
LIN {X 0,Y 401.779,Z 846.288,A -85,B 0,C 180,E1 15984.867,E2 15984.867} C_VEL
LIN {X 0,Y 399.576,Z 876.577,A -85,B 0,C 180,E1 15984.216,E2 15984.216} C_VEL
LIN {X 0,Y 396.941,Z 898.601,A -85,B 0,C 180,E1 15983.549,E2 15983.549} C_VEL
LIN {X 0,Y 393.388,Z 920.651,A -85,B 0,C 180,E1 15982.641,E2 15982.641} C_VEL
LIN {X 0,Y 389.342,Z 941.436,A -85,B 0,C 180,E1 15981.561,E2 15981.561} C_VEL
LIN {X 0,Y 384.398,Z 962.49,A -85,B 0,C 180,E1 15980.191,E2 15980.191} C_VEL
LIN {X 0,Y 379.129,Z 982.498,A -85,B 0,C 180,E1 15978.617,E2 15978.617} C_VEL
LIN {X 0,Y 373.313,Z 1001.857,A -85,B 0,C 180,E1 15976.762,E2 15976.762} C_VEL
LIN {X 0,Y 367.23,Z 1020.66,A -85,B 0,C 180,E1 15974.625,E2 15974.625} C_VEL
LIN {X 0,Y 361.489,Z 1037.116,A -85,B 0,C 180,E1 15972.395,E2 15972.395} C_VEL
LIN {X 0,Y 355.369,Z 1054.016,A -85,B 0,C 180,E1 15969.694,E2 15969.694} C_VEL
LIN {X 0,Y 349.841,Z 1068.83,A -85,B 0,C 180,E1 15966.884,E2 15966.884} C_VEL
LIN {X 0,Y 344.278,Z 1083.658,A -85,B 0,C 180,E1 15963.539,E2 15963.539} C_VEL
LIN {X 0,Y 339.774,Z 1096.099,A -85,B 0,C 180,E1 15960.213,E2 15960.213} C_VEL
LIN {X 0,Y 335.98,Z 1106.983,A -85,B 0,C 180,E1 15956.704,E2 15956.704} C_VEL
LIN {X 0,Y 332.946,Z 1116.731,A -85,B 0,C 180,E1 15952.98,E2 15952.98} C_VEL
LIN {X 0,Y 330.754,Z 1124.618,A -85,B 0,C 180,E1 15949.239,E2 15949.239} C_VEL
LIN {X 0,Y 329.273,Z 1131.345,A -85,B 0,C 180,E1 15945.319,E2 15945.319} C_VEL
LIN {X 0,Y 328.488,Z 1136.153,A -85,B 0,C 180,E1 15941.59,E2 15941.59} C_VEL
LIN {X 0,Y 328.085,Z 1139.84,A -85,B 0,C 180,E1 15937.707,E2 15937.707} C_VEL
LIN {X 0,Y 327.973,Z 1141.85,A -85,B 0,C 180,E1 15934.021,E2 15934.021} C_VEL
LIN {X 0,Y 327.95,Z 1142.247,A -85,B 0,C 180,E1 15932.966,E2 15932.966} C_VEL
LIN {X 0,Y 326.963,Z 1142.683,A -85,B 0,C 180,E1 15931.622,E2 15931.622} C_VEL
LIN {X 0,Y 322.862,Z 1142.994,A -85,B 0,C 180,E1 15929.362,E2 15929.362} C_VEL
LIN {X 0,Y 320.227,Z 1142.751,A -85,B 0,C 180,E1 15927.517,E2 15927.517} C_VEL
LIN {X 0,Y 319.956,Z 1142.53,A -85,B 0,C 180,E1 15926.817,E2 15926.817} C_VEL
LIN {X 0,Y 320.047,Z 1140.965,A -85,B 0,C 180,E1 15923.363,E2 15923.363} C_VEL
LIN {X 0,Y 320.3,Z 1138.238,A -85,B 0,C 180,E1 15919.751,E2 15919.751} C_VEL
LIN {X 0,Y 321.038,Z 1133.502,A -85,B 0,C 180,E1 15915.573,E2 15915.573} C_VEL
LIN {X 0,Y 322.307,Z 1127.748,A -85,B 0,C 180,E1 15911.741,E2 15911.741} C_VEL
LIN {X 0,Y 324.417,Z 1120.001,A -85,B 0,C 180,E1 15907.723,E2 15907.723} C_VEL
LIN {X 0,Y 327.36,Z 1110.994,A -85,B 0,C 180,E1 15903.893,E2 15903.893} C_VEL
LIN {X 0,Y 331.235,Z 1100.089,A -85,B 0,C 180,E1 15900.128,E2 15900.128} C_VEL
LIN {X 0,Y 335.927,Z 1087.904,A -85,B 0,C 180,E1 15896.589,E2 15896.589} C_VEL
LIN {X 0,Y 340.951,Z 1075.025,A -85,B 0,C 180,E1 15893.466,E2 15893.466} C_VEL
LIN {X 0,Y 347.149,Z 1059.319,A -85,B 0,C 180,E1 15890.253,E2 15890.253} C_VEL
LIN {X 0,Y 353.049,Z 1044.022,A -85,B 0,C 180,E1 15887.621,E2 15887.621} C_VEL
LIN {X 0,Y 359.546,Z 1026.34,A -85,B 0,C 180,E1 15885.062,E2 15885.062} C_VEL
LIN {X 0,Y 365.76,Z 1008.55,A -85,B 0,C 180,E1 15882.894,E2 15882.894} C_VEL
LIN {X 0,Y 371.652,Z 989.978,A -85,B 0,C 180,E1 15881.007,E2 15881.007} C_VEL
LIN {X 0,Y 377.405,Z 970.253,A -85,B 0,C 180,E1 15879.322,E2 15879.322} C_VEL
LIN {X 0,Y 382.596,Z 949.615,A -85,B 0,C 180,E1 15877.886,E2 15877.886} C_VEL
LIN {X 0,Y 387.193,Z 928.803,A -85,B 0,C 180,E1 15876.697,E2 15876.697} C_VEL
LIN {X 0,Y 390.966,Z 907.467,A -85,B 0,C 180,E1 15875.742,E2 15875.742} C_VEL
LIN {X 0,Y 394.129,Z 885.302,A -85,B 0,C 180,E1 15874.974,E2 15874.974} C_VEL
LIN {X 0,Y 396.273,Z 862.699,A -85,B 0,C 180,E1 15874.417,E2 15874.417} C_VEL
LIN {X 0,Y 408.177,Z 662.874,A -85,B 0,C 180,E1 15870.517,E2 15870.517} C_VEL
LIN {X 0,Y 409.089,Z 646.952,A -85,B 0,C 180,E1 15870.191,E2 15870.191} C_VEL
LIN {X 0,Y 401.432,Z 635.379,A -85,B 0,C 180,E1 15867.8,E2 15867.8} C_VEL
LIN {X 0,Y 392.994,Z 623.18,A -85,B 0,C 180,E1 15864.822,E2 15864.822} C_VEL
LIN {X 0,Y 385.349,Z 612.943,A -85,B 0,C 180,E1 15861.7,E2 15861.7} C_VEL
LIN {X 0,Y 380.932,Z 607.342,A -85,B 0,C 180,E1 15859.632,E2 15859.632} C_VEL
LIN {X 0,Y 376.963,Z 602.245,A -85,B 0,C 180,E1 15857.521,E2 15857.521} C_VEL
LIN {X 0,Y 373.545,Z 598.02,A -85,B 0,C 180,E1 15855.446,E2 15855.446} C_VEL
LIN {X 0,Y 372.556,Z 596.618,A -85,B 0,C 180,E1 15854.771,E2 15854.771} C_VEL
LIN {X 0,Y 369.458,Z 593.457,A -85,B 0,C 180,E1 15852.504,E2 15852.504} C_VEL
LIN {X 0,Y 367.973,Z 590.79,A -85,B 0,C 180,E1 15851.124,E2 15851.124} C_VEL
LIN {X 0,Y 364.561,Z 587.872,A -85,B 0,C 180,E1 15847.407,E2 15847.407} C_VEL
LIN {X 0,Y 363.169,Z 584.5,A -85,B 0,C 180,E1 15844.58,E2 15844.58} C_VEL
LIN {X 0,Y 362.779,Z 584.404,A -85,B 0,C 180,E1 15836.841,E2 15836.841} C_VEL
LIN {X 0,Y 363.332,Z 584.814,A -85,B 0,C 180,E1 15835.502,E2 15835.502} C_VEL
LIN {X 0,Y 365.133,Z 588.628,A -85,B 0,C 180,E1 15832.289,E2 15832.289} C_VEL
LIN {X 0,Y 368.23,Z 591.101,A -85,B 0,C 180,E1 15829.123,E2 15829.123} C_VEL
LIN {X 0,Y 370.81,Z 595.18,A -85,B 0,C 180,E1 15826.909,E2 15826.909} C_VEL
LIN {X 0,Y 373.189,Z 597.386,A -85,B 0,C 180,E1 15825.285,E2 15825.285} C_VEL
LIN {X 0,Y 376.443,Z 601.73,A -85,B 0,C 180,E1 15823.251,E2 15823.251} C_VEL
LIN {X 0,Y 377.892,Z 603.396,A -85,B 0,C 180,E1 15822.445,E2 15822.445} C_VEL
LIN {X 0,Y 381.69,Z 608.093,A -85,B 0,C 180,E1 15820.489,E2 15820.489} C_VEL
LIN {X 0,Y 386.967,Z 615.262,A -85,B 0,C 180,E1 15818.069,E2 15818.069} C_VEL
LIN {X 0,Y 392.292,Z 623.006,A -85,B 0,C 180,E1 15815.894,E2 15815.894} C_VEL
LIN {X 0,Y 399.599,Z 634.301,A -85,B 0,C 180,E1 15813.232,E2 15813.232} C_VEL
LIN {X 0,Y 408.266,Z 648.753,A -85,B 0,C 180,E1 15810.431,E2 15810.431} C_VEL
LIN {X 0,Y 409.241,Z 650.892,A -85,B 0,C 180,E1 15810.12,E2 15810.12} C_VEL
LIN {X 0,Y 396.703,Z 863.396,A -85,B 0,C 180,E1 15805.985,E2 15805.985} C_VEL
LIN {X 0,Y 394.414,Z 893.805,A -85,B 0,C 180,E1 15805.332,E2 15805.332} C_VEL
LIN {X 0,Y 391.575,Z 915.772,A -85,B 0,C 180,E1 15804.7,E2 15804.7} C_VEL
LIN {X 0,Y 387.696,Z 938.139,A -85,B 0,C 180,E1 15803.825,E2 15803.825} C_VEL
LIN {X 0,Y 383.57,Z 958.094,A -85,B 0,C 180,E1 15802.83,E2 15802.83} C_VEL
LIN {X 0,Y 378.275,Z 979.711,A -85,B 0,C 180,E1 15801.48,E2 15801.48} C_VEL
LIN {X 0,Y 372.797,Z 999.674,A -85,B 0,C 180,E1 15799.959,E2 15799.959} C_VEL
LIN {X 0,Y 366.653,Z 1019.547,A -85,B 0,C 180,E1 15798.113,E2 15798.113} C_VEL
LIN {X 0,Y 360.244,Z 1038.956,A -85,B 0,C 180,E1 15795.96,E2 15795.96} C_VEL
LIN {X 0,Y 354.108,Z 1056.202,A -85,B 0,C 180,E1 15793.659,E2 15793.659} C_VEL
LIN {X 0,Y 347.795,Z 1073.434,A -85,B 0,C 180,E1 15790.955,E2 15790.955} C_VEL
LIN {X 0,Y 342.006,Z 1088.792,A -85,B 0,C 180,E1 15788.087,E2 15788.087} C_VEL
LIN {X 0,Y 336.182,Z 1104.442,A -85,B 0,C 180,E1 15784.615,E2 15784.615} C_VEL
LIN {X 0,Y 331.589,Z 1117.268,A -85,B 0,C 180,E1 15781.241,E2 15781.241} C_VEL
LIN {X 0,Y 327.702,Z 1128.74,A -85,B 0,C 180,E1 15777.63,E2 15777.63} C_VEL
LIN {X 0,Y 324.631,Z 1139.05,A -85,B 0,C 180,E1 15773.796,E2 15773.796} C_VEL
LIN {X 0,Y 322.461,Z 1147.437,A -85,B 0,C 180,E1 15769.942,E2 15769.942} C_VEL
LIN {X 0,Y 321.028,Z 1154.644,A -85,B 0,C 180,E1 15765.907,E2 15765.907} C_VEL
LIN {X 0,Y 320.302,Z 1159.814,A -85,B 0,C 180,E1 15762.072,E2 15762.072} C_VEL
LIN {X 0,Y 320.018,Z 1163.652,A -85,B 0,C 180,E1 15758.263,E2 15758.263} C_VEL
LIN {X 0,Y 319.952,Z 1166.034,A -85,B 0,C 180,E1 15754.301,E2 15754.301} C_VEL
LIN {X 0,Y 319.949,Z 1166.884,A -85,B 0,C 180,E1 15751.074,E2 15751.074} C_VEL
LIN {X 0,Y 319.942,Z 1166.66,A -85,B 0,C 180,E1 15747.313,E2 15747.313} C_VEL
LIN {X 0,Y 319.965,Z 1164.892,A -85,B 0,C 180,E1 15743.54,E2 15743.54} C_VEL
LIN {X 0,Y 320.082,Z 1162.16,A -85,B 0,C 180,E1 15740.107,E2 15740.107} C_VEL
LIN {X 0,Y 320.576,Z 1157.528,A -85,B 0,C 180,E1 15736.104,E2 15736.104} C_VEL
LIN {X 0,Y 321.518,Z 1151.854,A -85,B 0,C 180,E1 15732.443,E2 15732.443} C_VEL
LIN {X 0,Y 323.271,Z 1144.045,A -85,B 0,C 180,E1 15728.403,E2 15728.403} C_VEL
LIN {X 0,Y 325.671,Z 1135.278,A -85,B 0,C 180,E1 15724.738,E2 15724.738} C_VEL
LIN {X 0,Y 329.327,Z 1123.785,A -85,B 0,C 180,E1 15720.737,E2 15720.737} C_VEL
LIN {X 0,Y 333.413,Z 1112.06,A -85,B 0,C 180,E1 15717.33,E2 15717.33} C_VEL
LIN {X 0,Y 338.67,Z 1097.662,A -85,B 0,C 180,E1 15713.809,E2 15713.809} C_VEL
LIN {X 0,Y 344.311,Z 1082.736,A -85,B 0,C 180,E1 15710.723,E2 15710.723} C_VEL
LIN {X 0,Y 350.367,Z 1066.33,A -85,B 0,C 180,E1 15707.883,E2 15707.883} C_VEL
LIN {X 0,Y 356.79,Z 1048.731,A -85,B 0,C 180,E1 15705.299,E2 15705.299} C_VEL
LIN {X 0,Y 362.93,Z 1030.844,A -85,B 0,C 180,E1 15703.107,E2 15703.107} C_VEL
LIN {X 0,Y 369.264,Z 1011.242,A -85,B 0,C 180,E1 15701.081,E2 15701.081} C_VEL
LIN {X 0,Y 374.855,Z 992.196,A -85,B 0,C 180,E1 15699.448,E2 15699.448} C_VEL
LIN {X 0,Y 380.656,Z 970.12,A -85,B 0,C 180,E1 15697.89,E2 15697.89} C_VEL
LIN {X 0,Y 385.396,Z 949.35,A -85,B 0,C 180,E1 15696.71,E2 15696.71} C_VEL
LIN {X 0,Y 389.799,Z 926.055,A -85,B 0,C 180,E1 15695.675,E2 15695.675} C_VEL
LIN {X 0,Y 393.297,Z 903.18,A -85,B 0,C 180,E1 15694.914,E2 15694.914} C_VEL
LIN {X 0,Y 395.613,Z 879.608,A -85,B 0,C 180,E1 15694.348,E2 15694.348} C_VEL
LIN {X 0,Y 407.271,Z 681.626,A -85,B 0,C 180,E1 15690.48,E2 15690.48} C_VEL
LIN {X 0,Y 409.129,Z 650.447,A -85,B 0,C 180,E1 15689.863,E2 15689.863} C_VEL
LIN {X 0,Y 401.064,Z 636.801,A -85,B 0,C 180,E1 15687.304,E2 15687.304} C_VEL
LIN {X 0,Y 393.895,Z 625.424,A -85,B 0,C 180,E1 15684.761,E2 15684.761} C_VEL
LIN {X 0,Y 387.912,Z 616.592,A -85,B 0,C 180,E1 15682.385,E2 15682.385} C_VEL
LIN {X 0,Y 384.588,Z 612.141,A -85,B 0,C 180,E1 15680.945,E2 15680.945} C_VEL
LIN {X 0,Y 380.956,Z 607.414,A -85,B 0,C 180,E1 15679.231,E2 15679.231} C_VEL
LIN {X 0,Y 376.834,Z 602.105,A -85,B 0,C 180,E1 15677.049,E2 15677.049} C_VEL
LIN {X 0,Y 373.408,Z 597.848,A -85,B 0,C 180,E1 15674.974,E2 15674.974} C_VEL
LIN {X 0,Y 372.638,Z 596.705,A -85,B 0,C 180,E1 15674.45,E2 15674.45} C_VEL
LIN {X 0,Y 369.395,Z 593.42,A -85,B 0,C 180,E1 15672.109,E2 15672.109} C_VEL
LIN {X 0,Y 367.806,Z 590.664,A -85,B 0,C 180,E1 15670.652,E2 15670.652} C_VEL
LIN {X 0,Y 364.386,Z 587.629,A -85,B 0,C 180,E1 15666.934,E2 15666.934} C_VEL
LIN {X 0,Y 363.107,Z 584.492,A -85,B 0,C 180,E1 15664.422,E2 15664.422} C_VEL
LIN {X 0,Y 362.316,Z 584.277,A -85,B 0,C 180,E1 15656.994,E2 15656.994} C_VEL
LIN {X 0,Y 363.237,Z 584.733,A -85,B 0,C 180,E1 15654.709,E2 15654.709} C_VEL
LIN {X 0,Y 365.124,Z 588.617,A -85,B 0,C 180,E1 15651.496,E2 15651.496} C_VEL
LIN {X 0,Y 368.208,Z 591.16,A -85,B 0,C 180,E1 15648.407,E2 15648.407} C_VEL
LIN {X 0,Y 370.733,Z 595.128,A -85,B 0,C 180,E1 15646.27,E2 15646.27} C_VEL
LIN {X 0,Y 373.065,Z 597.227,A -85,B 0,C 180,E1 15644.693,E2 15644.693} C_VEL
LIN {X 0,Y 376.272,Z 601.632,A -85,B 0,C 180,E1 15642.685,E2 15642.685} C_VEL
LIN {X 0,Y 377.863,Z 603.43,A -85,B 0,C 180,E1 15641.806,E2 15641.806} C_VEL
LIN {X 0,Y 382.416,Z 609.243,A -85,B 0,C 180,E1 15639.491,E2 15639.491} C_VEL
LIN {X 0,Y 386.733,Z 614.97,A -85,B 0,C 180,E1 15637.543,E2 15637.543} C_VEL
LIN {X 0,Y 391.513,Z 621.378,A -85,B 0,C 180,E1 15635.601,E2 15635.601} C_VEL
LIN {X 0,Y 397.6,Z 629.909,A -85,B 0,C 180,E1 15633.368,E2 15633.368} C_VEL
LIN {X 0,Y 405.719,Z 641.768,A -85,B 0,C 180,E1 15630.713,E2 15630.713} C_VEL
LIN {X 0,Y 409.066,Z 647.288,A -85,B 0,C 180,E1 15629.688,E2 15629.688} C_VEL
LIN {X 0,Y 397.077,Z 849.279,A -85,B 0,C 180,E1 15625.759,E2 15625.759} C_VEL
LIN {X 0,Y 394.898,Z 877.38,A -85,B 0,C 180,E1 15625.145,E2 15625.145} C_VEL
LIN {X 0,Y 392.101,Z 899.939,A -85,B 0,C 180,E1 15624.456,E2 15624.456} C_VEL
LIN {X 0,Y 388.414,Z 921.772,A -85,B 0,C 180,E1 15623.545,E2 15623.545} C_VEL
LIN {X 0,Y 384.123,Z 942.995,A -85,B 0,C 180,E1 15622.43,E2 15622.43} C_VEL
LIN {X 0,Y 379.103,Z 963.444,A -85,B 0,C 180,E1 15621.083,E2 15621.083} C_VEL
LIN {X 0,Y 373.561,Z 983.617,A -85,B 0,C 180,E1 15619.478,E2 15619.478} C_VEL
LIN {X 0,Y 367.779,Z 1002.168,A -85,B 0,C 180,E1 15617.687,E2 15617.687} C_VEL
LIN {X 0,Y 361.457,Z 1020.971,A -85,B 0,C 180,E1 15615.536,E2 15615.536} C_VEL
LIN {X 0,Y 355.567,Z 1037.166,A -85,B 0,C 180,E1 15613.325,E2 15613.325} C_VEL
LIN {X 0,Y 349.062,Z 1054.329,A -85,B 0,C 180,E1 15610.559,E2 15610.559} C_VEL
LIN {X 0,Y 343.271,Z 1069.142,A -85,B 0,C 180,E1 15607.711,E2 15607.711} C_VEL
LIN {X 0,Y 337.615,Z 1083.447,A -85,B 0,C 180,E1 15604.448,E2 15604.448} C_VEL
LIN {X 0,Y 332.872,Z 1095.789,A -85,B 0,C 180,E1 15601.108,E2 15601.108} C_VEL
LIN {X 0,Y 328.613,Z 1107.295,A -85,B 0,C 180,E1 15597.352,E2 15597.352} C_VEL
LIN {X 0,Y 325.369,Z 1117.042,A -85,B 0,C 180,E1 15593.547,E2 15593.547} C_VEL
LIN {X 0,Y 323.017,Z 1124.927,A -85,B 0,C 180,E1 15589.719,E2 15589.719} C_VEL
LIN {X 0,Y 321.413,Z 1131.652,A -85,B 0,C 180,E1 15585.703,E2 15585.703} C_VEL
LIN {X 0,Y 320.548,Z 1136.458,A -85,B 0,C 180,E1 15581.881,E2 15581.881} C_VEL
LIN {X 0,Y 320.115,Z 1140.142,A -85,B 0,C 180,E1 15577.9,E2 15577.9} C_VEL
LIN {X 0,Y 319.983,Z 1142.151,A -85,B 0,C 180,E1 15574.122,E2 15574.122} C_VEL
LIN {X 0,Y 319.946,Z 1142.93,A -85,B 0,C 180,E1 15570.717,E2 15570.717} C_VEL
LIN {X 0,Y 319.956,Z 1142.53,A -85,B 0,C 180,E1 15566.817,E2 15566.817} C_VEL
LIN {X 0,Y 318.981,Z 1142.078,A -85,B 0,C 180,E1 15565.44,E2 15565.44} C_VEL
LIN {X 0,Y 314.799,Z 1141.06,A -85,B 0,C 180,E1 15563.029,E2 15563.029} C_VEL
LIN {X 0,Y 312.467,Z 1139.986,A -85,B 0,C 180,E1 15561.244,E2 15561.244} C_VEL
LIN {X 0,Y 312.252,Z 1139.407,A -85,B 0,C 180,E1 15560.533,E2 15560.533} C_VEL
LIN {X 0,Y 312.803,Z 1135.669,A -85,B 0,C 180,E1 15556.695,E2 15556.695} C_VEL
LIN {X 0,Y 313.999,Z 1130.111,A -85,B 0,C 180,E1 15552.583,E2 15552.583} C_VEL
LIN {X 0,Y 315.89,Z 1123.352,A -85,B 0,C 180,E1 15548.654,E2 15548.654} C_VEL
LIN {X 0,Y 318.796,Z 1114.469,A -85,B 0,C 180,E1 15544.553,E2 15544.553} C_VEL
LIN {X 0,Y 322.598,Z 1104.319,A -85,B 0,C 180,E1 15540.679,E2 15540.679} C_VEL
LIN {X 0,Y 327.187,Z 1092.668,A -85,B 0,C 180,E1 15537.047,E2 15537.047} C_VEL
LIN {X 0,Y 332.799,Z 1079.116,A -85,B 0,C 180,E1 15533.497,E2 15533.497} C_VEL
LIN {X 0,Y 338.627,Z 1065.008,A -85,B 0,C 180,E1 15530.413,E2 15530.413} C_VEL
LIN {X 0,Y 345.417,Z 1048.323,A -85,B 0,C 180,E1 15527.364,E2 15527.364} C_VEL
LIN {X 0,Y 351.628,Z 1032.505,A -85,B 0,C 180,E1 15524.925,E2 15524.925} C_VEL
LIN {X 0,Y 358.352,Z 1014.134,A -85,B 0,C 180,E1 15522.557,E2 15522.557} C_VEL
LIN {X 0,Y 364.868,Z 995.128,A -85,B 0,C 180,E1 15520.501,E2 15520.501} C_VEL
LIN {X 0,Y 370.903,Z 975.295,A -85,B 0,C 180,E1 15518.74,E2 15518.74} C_VEL
LIN {X 0,Y 376.601,Z 954.399,A -85,B 0,C 180,E1 15517.204,E2 15517.204} C_VEL
LIN {X 0,Y 381.289,Z 934.239,A -85,B 0,C 180,E1 15516.003,E2 15516.003} C_VEL
LIN {X 0,Y 385.831,Z 910.779,A -85,B 0,C 180,E1 15514.896,E2 15514.896} C_VEL
LIN {X 0,Y 388.957,Z 890.18,A -85,B 0,C 180,E1 15514.149,E2 15514.149} C_VEL
LIN {X 0,Y 391.564,Z 866.048,A -85,B 0,C 180,E1 15513.518,E2 15513.518} C_VEL
LIN {X 0,Y 403.316,Z 676.486,A -85,B 0,C 180,E1 15509.797,E2 15509.797} C_VEL
LIN {X 0,Y 404.9,Z 651.485,A -85,B 0,C 180,E1 15509.308,E2 15509.308} C_VEL
LIN {X 0,Y 396.819,Z 639.185,A -85,B 0,C 180,E1 15506.648,E2 15506.648} C_VEL
LIN {X 0,Y 389.423,Z 628.631,A -85,B 0,C 180,E1 15503.893,E2 15503.893} C_VEL
LIN {X 0,Y 383.418,Z 620.316,A -85,B 0,C 180,E1 15501.333,E2 15501.333} C_VEL
LIN {X 0,Y 379.089,Z 614.738,A -85,B 0,C 180,E1 15499.25,E2 15499.25} C_VEL
LIN {X 0,Y 375.208,Z 609.7,A -85,B 0,C 180,E1 15497.126,E2 15497.126} C_VEL
LIN {X 0,Y 371.896,Z 605.384,A -85,B 0,C 180,E1 15495.037,E2 15495.037} C_VEL
LIN {X 0,Y 370.915,Z 604.183,A -85,B 0,C 180,E1 15494.36,E2 15494.36} C_VEL
LIN {X 0,Y 367.858,Z 600.72,A -85,B 0,C 180,E1 15492.001,E2 15492.001} C_VEL
LIN {X 0,Y 366.66,Z 598.595,A -85,B 0,C 180,E1 15490.846,E2 15490.846} C_VEL
LIN {X 0,Y 363.377,Z 595.589,A -85,B 0,C 180,E1 15487.113,E2 15487.113} C_VEL
LIN {X 0,Y 362.124,Z 592.426,A -85,B 0,C 180,E1 15484.434,E2 15484.434} C_VEL
LIN {X 0,Y 361.864,Z 592.363,A -85,B 0,C 180,E1 15476.674,E2 15476.674} C_VEL
LIN {X 0,Y 362.28,Z 592.739,A -85,B 0,C 180,E1 15475.648,E2 15475.648} C_VEL
LIN {X 0,Y 364.157,Z 596.647,A -85,B 0,C 180,E1 15472.268,E2 15472.268} C_VEL
LIN {X 0,Y 366.991,Z 598.994,A -85,B 0,C 180,E1 15469.324,E2 15469.324} C_VEL
LIN {X 0,Y 369.635,Z 603.087,A -85,B 0,C 180,E1 15467.026,E2 15467.026} C_VEL
LIN {X 0,Y 371.692,Z 605.015,A -85,B 0,C 180,E1 15465.592,E2 15465.592} C_VEL
LIN {X 0,Y 375.088,Z 609.54,A -85,B 0,C 180,E1 15463.428,E2 15463.428} C_VEL
LIN {X 0,Y 376.563,Z 611.487,A -85,B 0,C 180,E1 15462.58,E2 15462.58} C_VEL
LIN {X 0,Y 380.755,Z 616.907,A -85,B 0,C 180,E1 15460.399,E2 15460.399} C_VEL
LIN {X 0,Y 384.828,Z 622.378,A -85,B 0,C 180,E1 15458.51,E2 15458.51} C_VEL
LIN {X 0,Y 390.058,Z 630.157,A -85,B 0,C 180,E1 15456.309,E2 15456.309} C_VEL
LIN {X 0,Y 397.04,Z 641.195,A -85,B 0,C 180,E1 15453.691,E2 15453.691} C_VEL
LIN {X 0,Y 405.022,Z 654.833,A -85,B 0,C 180,E1 15451.025,E2 15451.025} C_VEL
LIN {X 0,Y 391.996,Z 867.559,A -85,B 0,C 180,E1 15446.873,E2 15446.873} C_VEL
LIN {X 0,Y 389.799,Z 894.332,A -85,B 0,C 180,E1 15446.284,E2 15446.284} C_VEL
LIN {X 0,Y 386.709,Z 917.294,A -85,B 0,C 180,E1 15445.617,E2 15445.617} C_VEL
LIN {X 0,Y 382.804,Z 938.701,A -85,B 0,C 180,E1 15444.764,E2 15444.764} C_VEL
LIN {X 0,Y 378.229,Z 959.997,A -85,B 0,C 180,E1 15443.691,E2 15443.691} C_VEL
LIN {X 0,Y 372.69,Z 981.434,A -85,B 0,C 180,E1 15442.319,E2 15442.319} C_VEL
LIN {X 0,Y 366.806,Z 1001.849,A -85,B 0,C 180,E1 15440.727,E2 15440.727} C_VEL
LIN {X 0,Y 360.684,Z 1020.784,A -85,B 0,C 180,E1 15438.93,E2 15438.93} C_VEL
LIN {X 0,Y 353.836,Z 1040.494,A -85,B 0,C 180,E1 15436.688,E2 15436.688} C_VEL
LIN {X 0,Y 347.503,Z 1057.579,A -85,B 0,C 180,E1 15434.361,E2 15434.361} C_VEL
LIN {X 0,Y 340.575,Z 1075.473,A -85,B 0,C 180,E1 15431.454,E2 15431.454} C_VEL
LIN {X 0,Y 334.458,Z 1091.083,A -85,B 0,C 180,E1 15428.442,E2 15428.442} C_VEL
LIN {X 0,Y 328.749,Z 1105.557,A -85,B 0,C 180,E1 15425.087,E2 15425.087} C_VEL
LIN {X 0,Y 323.759,Z 1118.799,A -85,B 0,C 180,E1 15421.461,E2 15421.461} C_VEL
LIN {X 0,Y 319.768,Z 1130.022,A -85,B 0,C 180,E1 15417.763,E2 15417.763} C_VEL
LIN {X 0,Y 316.373,Z 1140.834,A -85,B 0,C 180,E1 15413.466,E2 15413.466} C_VEL
LIN {X 0,Y 314.256,Z 1148.944,A -85,B 0,C 180,E1 15409.516,E2 15409.516} C_VEL
LIN {X 0,Y 312.883,Z 1155.651,A -85,B 0,C 180,E1 15405.381,E2 15405.381} C_VEL
LIN {X 0,Y 312.251,Z 1160.363,A -85,B 0,C 180,E1 15401.638,E2 15401.638} C_VEL
LIN {X 0,Y 311.971,Z 1164.002,A -85,B 0,C 180,E1 15397.55,E2 15397.55} C_VEL
LIN {X 0,Y 311.954,Z 1165.875,A -85,B 0,C 180,E1 15394.043,E2 15394.043} C_VEL
LIN {X 0,Y 311.952,Z 1166.677,A -85,B 0,C 180,E1 15390.367,E2 15390.367} C_VEL
LIN {X 0,Y 311.94,Z 1166.084,A -85,B 0,C 180,E1 15386.508,E2 15386.508} C_VEL
LIN {X 0,Y 311.961,Z 1164.354,A -85,B 0,C 180,E1 15383.004,E2 15383.004} C_VEL
LIN {X 0,Y 312.151,Z 1161.357,A -85,B 0,C 180,E1 15379.293,E2 15379.293} C_VEL
LIN {X 0,Y 312.753,Z 1156.433,A -85,B 0,C 180,E1 15375.181,E2 15375.181} C_VEL
LIN {X 0,Y 313.866,Z 1150.606,A -85,B 0,C 180,E1 15371.423,E2 15371.423} C_VEL
LIN {X 0,Y 315.901,Z 1142.485,A -85,B 0,C 180,E1 15367.285,E2 15367.285} C_VEL
LIN {X 0,Y 318.754,Z 1133.148,A -85,B 0,C 180,E1 15363.377,E2 15363.377} C_VEL
LIN {X 0,Y 322.661,Z 1121.71,A -85,B 0,C 180,E1 15359.455,E2 15359.455} C_VEL
LIN {X 0,Y 327.397,Z 1109.095,A -85,B 0,C 180,E1 15355.81,E2 15355.81} C_VEL
LIN {X 0,Y 332.869,Z 1094.992,A -85,B 0,C 180,E1 15352.427,E2 15352.427} C_VEL
LIN {X 0,Y 339.418,Z 1078.343,A -85,B 0,C 180,E1 15349.07,E2 15349.07} C_VEL
LIN {X 0,Y 345.851,Z 1061.902,A -85,B 0,C 180,E1 15346.294,E2 15346.294} C_VEL
LIN {X 0,Y 352.403,Z 1044.307,A -85,B 0,C 180,E1 15343.811,E2 15343.811} C_VEL
LIN {X 0,Y 359.004,Z 1025.795,A -85,B 0,C 180,E1 15341.599,E2 15341.599} C_VEL
LIN {X 0,Y 365.507,Z 1005.735,A -85,B 0,C 180,E1 15339.628,E2 15339.628} C_VEL
LIN {X 0,Y 371.856,Z 984.319,A -85,B 0,C 180,E1 15337.891,E2 15337.891} C_VEL
LIN {X 0,Y 377.144,Z 964.004,A -85,B 0,C 180,E1 15336.553,E2 15336.553} C_VEL
LIN {X 0,Y 382.217,Z 941.315,A -85,B 0,C 180,E1 15335.36,E2 15335.36} C_VEL
LIN {X 0,Y 386.116,Z 920.243,A -85,B 0,C 180,E1 15334.496,E2 15334.496} C_VEL
LIN {X 0,Y 389.466,Z 896.65,A -85,B 0,C 180,E1 15333.782,E2 15333.782} C_VEL
LIN {X 0,Y 391.608,Z 872.96,A -85,B 0,C 180,E1 15333.239,E2 15333.239} C_VEL
LIN {X 0,Y 404.335,Z 664.252,A -85,B 0,C 180,E1 15329.165,E2 15329.165} C_VEL
LIN {X 0,Y 404.852,Z 654.541,A -85,B 0,C 180,E1 15328.95,E2 15328.95} C_VEL
LIN {X 0,Y 395.914,Z 639.394,A -85,B 0,C 180,E1 15325.946,E2 15325.946} C_VEL
LIN {X 0,Y 388.168,Z 627.238,A -85,B 0,C 180,E1 15322.969,E2 15322.969} C_VEL
LIN {X 0,Y 382.823,Z 619.687,A -85,B 0,C 180,E1 15320.646,E2 15320.646} C_VEL
LIN {X 0,Y 379.105,Z 614.807,A -85,B 0,C 180,E1 15318.849,E2 15318.849} C_VEL
LIN {X 0,Y 375.207,Z 609.675,A -85,B 0,C 180,E1 15316.726,E2 15316.726} C_VEL
LIN {X 0,Y 371.755,Z 605.209,A -85,B 0,C 180,E1 15314.564,E2 15314.564} C_VEL
LIN {X 0,Y 370.537,Z 603.923,A -85,B 0,C 180,E1 15313.736,E2 15313.736} C_VEL
LIN {X 0,Y 367.535,Z 600.231,A -85,B 0,C 180,E1 15311.375,E2 15311.375} C_VEL
LIN {X 0,Y 366.666,Z 598.547,A -85,B 0,C 180,E1 15310.527,E2 15310.527} C_VEL
LIN {X 0,Y 363.3,Z 595.513,A -85,B 0,C 180,E1 15306.796,E2 15306.796} C_VEL
LIN {X 0,Y 362.056,Z 592.417,A -85,B 0,C 180,E1 15304.276,E2 15304.276} C_VEL
LIN {X 0,Y 361.389,Z 592.236,A -85,B 0,C 180,E1 15296.828,E2 15296.828} C_VEL
LIN {X 0,Y 362.181,Z 592.667,A -85,B 0,C 180,E1 15294.852,E2 15294.852} C_VEL
LIN {X 0,Y 364.025,Z 596.497,A -85,B 0,C 180,E1 15291.629,E2 15291.629} C_VEL
LIN {X 0,Y 366.891,Z 598.885,A -85,B 0,C 180,E1 15288.684,E2 15288.684} C_VEL
LIN {X 0,Y 369.456,Z 602.931,A -85,B 0,C 180,E1 15286.461,E2 15286.461} C_VEL
LIN {X 0,Y 371.631,Z 604.988,A -85,B 0,C 180,E1 15284.952,E2 15284.952} C_VEL
LIN {X 0,Y 374.919,Z 609.447,A -85,B 0,C 180,E1 15282.861,E2 15282.861} C_VEL
LIN {X 0,Y 376.344,Z 611.211,A -85,B 0,C 180,E1 15282.05,E2 15282.05} C_VEL
LIN {X 0,Y 380.684,Z 616.837,A -85,B 0,C 180,E1 15279.795,E2 15279.795} C_VEL
LIN {X 0,Y 384.772,Z 622.348,A -85,B 0,C 180,E1 15277.905,E2 15277.905} C_VEL
LIN {X 0,Y 390.981,Z 630.733,A -85,B 0,C 180,E1 15275.364,E2 15275.364} C_VEL
LIN {X 0,Y 400.327,Z 644.462,A -85,B 0,C 180,E1 15272.035,E2 15272.035} C_VEL
LIN {X 0,Y 404.825,Z 651.63,A -85,B 0,C 180,E1 15270.588,E2 15270.588} C_VEL
LIN {X 0,Y 392.472,Z 852.294,A -85,B 0,C 180,E1 15266.671,E2 15266.671} C_VEL
LIN {X 0,Y 390.325,Z 878.183,A -85,B 0,C 180,E1 15266.096,E2 15266.096} C_VEL
LIN {X 0,Y 387.388,Z 901.023,A -85,B 0,C 180,E1 15265.393,E2 15265.393} C_VEL
LIN {X 0,Y 383.581,Z 922.672,A -85,B 0,C 180,E1 15264.482,E2 15264.482} C_VEL
LIN {X 0,Y 378.983,Z 944.436,A -85,B 0,C 180,E1 15263.326,E2 15263.326} C_VEL
LIN {X 0,Y 374.073,Z 963.755,A -85,B 0,C 180,E1 15262.047,E2 15262.047} C_VEL
LIN {X 0,Y 368.337,Z 983.927,A -85,B 0,C 180,E1 15260.438,E2 15260.438} C_VEL
LIN {X 0,Y 362.342,Z 1002.479,A -85,B 0,C 180,E1 15258.64,E2 15258.64} C_VEL
LIN {X 0,Y 355.778,Z 1021.282,A -85,B 0,C 180,E1 15256.476,E2 15256.476} C_VEL
LIN {X 0,Y 349.489,Z 1037.881,A -85,B 0,C 180,E1 15254.188,E2 15254.188} C_VEL
LIN {X 0,Y 342.464,Z 1055.553,A -85,B 0,C 180,E1 15251.288,E2 15251.288} C_VEL
LIN {X 0,Y 336.443,Z 1070.286,A -85,B 0,C 180,E1 15248.398,E2 15248.398} C_VEL
LIN {X 0,Y 330.536,Z 1084.447,A -85,B 0,C 180,E1 15245.082,E2 15245.082} C_VEL
LIN {X 0,Y 325.34,Z 1097.324,A -85,B 0,C 180,E1 15241.498,E2 15241.498} C_VEL
LIN {X 0,Y 320.917,Z 1108.613,A -85,B 0,C 180,E1 15237.661,E2 15237.661} C_VEL
LIN {X 0,Y 317.268,Z 1118.928,A -85,B 0,C 180,E1 15233.397,E2 15233.397} C_VEL
LIN {X 0,Y 314.901,Z 1126.683,A -85,B 0,C 180,E1 15229.434,E2 15229.434} C_VEL
LIN {X 0,Y 313.325,Z 1132.943,A -85,B 0,C 180,E1 15225.359,E2 15225.359} C_VEL
LIN {X 0,Y 312.499,Z 1137.562,A -85,B 0,C 180,E1 15221.442,E2 15221.442} C_VEL
LIN {X 0,Y 312.079,Z 1140.881,A -85,B 0,C 180,E1 15217.363,E2 15217.363} C_VEL
LIN {X 0,Y 311.98,Z 1142.583,A -85,B 0,C 180,E1 15213.859,E2 15213.859} C_VEL
LIN {X 0,Y 311.97,Z 1143.317,A -85,B 0,C 180,E1 15210,E2 15210} C_VEL
LIN {X 0,Y 311.978,Z 1142.617,A -85,B 0,C 180,E1 15206.141,E2 15206.141} C_VEL
LIN {X 0,Y 312.075,Z 1140.939,A -85,B 0,C 180,E1 15202.637,E2 15202.637} C_VEL
LIN {X 0,Y 312.252,Z 1139.407,A -85,B 0,C 180,E1 15200.533,E2 15200.533} C_VEL
LIN {X 0,Y 311.403,Z 1138.324,A -85,B 0,C 180,E1 15199.132,E2 15199.132} C_VEL
LIN {X 0,Y 305.777,Z 1134.659,A -85,B 0,C 180,E1 15195.268,E2 15195.268} C_VEL
LIN {X 0,Y 305.467,Z 1133.26,A -85,B 0,C 180,E1 15194.147,E2 15194.147} C_VEL
LIN {X 0,Y 307.352,Z 1126.405,A -85,B 0,C 180,E1 15189.63,E2 15189.63} C_VEL
LIN {X 0,Y 309.802,Z 1119.038,A -85,B 0,C 180,E1 15185.803,E2 15185.803} C_VEL
LIN {X 0,Y 313.535,Z 1109.164,A -85,B 0,C 180,E1 15181.631,E2 15181.631} C_VEL
LIN {X 0,Y 317.957,Z 1098.463,A -85,B 0,C 180,E1 15177.897,E2 15177.897} C_VEL
LIN {X 0,Y 323.381,Z 1085.772,A -85,B 0,C 180,E1 15174.242,E2 15174.242} C_VEL
LIN {X 0,Y 329.536,Z 1071.818,A -85,B 0,C 180,E1 15170.869,E2 15170.869} C_VEL
LIN {X 0,Y 335.781,Z 1057.196,A -85,B 0,C 180,E1 15167.934,E2 15167.934} C_VEL
LIN {X 0,Y 342.79,Z 1040.478,A -85,B 0,C 180,E1 15165.1,E2 15165.1} C_VEL
LIN {X 0,Y 349.319,Z 1023.941,A -85,B 0,C 180,E1 15162.762,E2 15162.762} C_VEL
LIN {X 0,Y 356.595,Z 1004.17,A -85,B 0,C 180,E1 15160.425,E2 15160.425} C_VEL
LIN {X 0,Y 362.515,Z 986.555,A -85,B 0,C 180,E1 15158.69,E2 15158.69} C_VEL
LIN {X 0,Y 368.815,Z 965.534,A -85,B 0,C 180,E1 15156.973,E2 15156.973} C_VEL
LIN {X 0,Y 374.065,Z 945.627,A -85,B 0,C 180,E1 15155.641,E2 15155.641} C_VEL
LIN {X 0,Y 378.933,Z 923.508,A -85,B 0,C 180,E1 15154.456,E2 15154.456} C_VEL
LIN {X 0,Y 382.926,Z 901.564,A -85,B 0,C 180,E1 15153.53,E2 15153.53} C_VEL
LIN {X 0,Y 385.967,Z 878.748,A -85,B 0,C 180,E1 15152.828,E2 15152.828} C_VEL
LIN {X 0,Y 388.174,Z 853.233,A -85,B 0,C 180,E1 15152.257,E2 15152.257} C_VEL
LIN {X 0,Y 400.765,Z 656.072,A -85,B 0,C 180,E1 15148.397,E2 15148.397} C_VEL
LIN {X 0,Y 393.628,Z 645.137,A -85,B 0,C 180,E1 15145.943,E2 15145.943} C_VEL
LIN {X 0,Y 386.972,Z 635.416,A -85,B 0,C 180,E1 15143.367,E2 15143.367} C_VEL
LIN {X 0,Y 380.883,Z 626.965,A -85,B 0,C 180,E1 15140.676,E2 15140.676} C_VEL
LIN {X 0,Y 377.405,Z 622.284,A -85,B 0,C 180,E1 15138.938,E2 15138.938} C_VEL
LIN {X 0,Y 373.473,Z 617.146,A -85,B 0,C 180,E1 15136.727,E2 15136.727} C_VEL
LIN {X 0,Y 370.165,Z 612.556,A -85,B 0,C 180,E1 15134.549,E2 15134.549} C_VEL
LIN {X 0,Y 366.531,Z 608.414,A -85,B 0,C 180,E1 15131.726,E2 15131.726} C_VEL
LIN {X 0,Y 365.526,Z 606.48,A -85,B 0,C 180,E1 15130.72,E2 15130.72} C_VEL
LIN {X 0,Y 362.202,Z 603.304,A -85,B 0,C 180,E1 15126.818,E2 15126.818} C_VEL
LIN {X 0,Y 361.082,Z 600.351,A -85,B 0,C 180,E1 15124.288,E2 15124.288} C_VEL
LIN {X 0,Y 360.952,Z 600.323,A -85,B 0,C 180,E1 15116.507,E2 15116.507} C_VEL
LIN {X 0,Y 361.257,Z 600.773,A -85,B 0,C 180,E1 15115.715,E2 15115.715} C_VEL
LIN {X 0,Y 363.182,Z 604.662,A -85,B 0,C 180,E1 15112.248,E2 15112.248} C_VEL
LIN {X 0,Y 365.686,Z 606.706,A -85,B 0,C 180,E1 15109.604,E2 15109.604} C_VEL
LIN {X 0,Y 368.361,Z 610.887,A -85,B 0,C 180,E1 15107.22,E2 15107.22} C_VEL
LIN {X 0,Y 370.372,Z 612.943,A -85,B 0,C 180,E1 15105.779,E2 15105.779} C_VEL
LIN {X 0,Y 373.867,Z 617.469,A -85,B 0,C 180,E1 15103.532,E2 15103.532} C_VEL
LIN {X 0,Y 379.035,Z 624.486,A -85,B 0,C 180,E1 15100.708,E2 15100.708} C_VEL
LIN {X 0,Y 383.117,Z 630.095,A -85,B 0,C 180,E1 15098.771,E2 15098.771} C_VEL
LIN {X 0,Y 387.929,Z 637.443,A -85,B 0,C 180,E1 15096.695,E2 15096.695} C_VEL
LIN {X 0,Y 394.506,Z 648.087,A -85,B 0,C 180,E1 15094.156,E2 15094.156} C_VEL
LIN {X 0,Y 400.871,Z 659.278,A -85,B 0,C 180,E1 15091.939,E2 15091.939} C_VEL
LIN {X 0,Y 387.407,Z 871.364,A -85,B 0,C 180,E1 15087.789,E2 15087.789} C_VEL
LIN {X 0,Y 385.218,Z 895.51,A -85,B 0,C 180,E1 15087.242,E2 15087.242} C_VEL
LIN {X 0,Y 381.913,Z 918.665,A -85,B 0,C 180,E1 15086.555,E2 15086.555} C_VEL
LIN {X 0,Y 377.869,Z 939.98,A -85,B 0,C 180,E1 15085.695,E2 15085.695} C_VEL
LIN {X 0,Y 372.973,Z 961.612,A -85,B 0,C 180,E1 15084.583,E2 15084.583} C_VEL
LIN {X 0,Y 367.759,Z 981.134,A -85,B 0,C 180,E1 15083.326,E2 15083.326} C_VEL
LIN {X 0,Y 361.67,Z 1001.546,A -85,B 0,C 180,E1 15081.733,E2 15081.733} C_VEL
LIN {X 0,Y 355.343,Z 1020.421,A -85,B 0,C 180,E1 15079.938,E2 15079.938} C_VEL
LIN {X 0,Y 348.197,Z 1040.187,A -85,B 0,C 180,E1 15077.682,E2 15077.682} C_VEL
LIN {X 0,Y 341.591,Z 1057.27,A -85,B 0,C 180,E1 15075.339,E2 15075.339} C_VEL
LIN {X 0,Y 334.558,Z 1074.692,A -85,B 0,C 180,E1 15072.487,E2 15072.487} C_VEL
LIN {X 0,Y 328.284,Z 1089.887,A -85,B 0,C 180,E1 15069.535,E2 15069.535} C_VEL
LIN {X 0,Y 322.21,Z 1104.53,A -85,B 0,C 180,E1 15066.128,E2 15066.128} C_VEL
LIN {X 0,Y 317.114,Z 1117.289,A -85,B 0,C 180,E1 15062.626,E2 15062.626} C_VEL
LIN {X 0,Y 312.74,Z 1128.713,A -85,B 0,C 180,E1 15058.837,E2 15058.837} C_VEL
LIN {X 0,Y 309.3,Z 1138.857,A -85,B 0,C 180,E1 15054.85,E2 15054.85} C_VEL
LIN {X 0,Y 306.796,Z 1147.343,A -85,B 0,C 180,E1 15050.718,E2 15050.718} C_VEL
LIN {X 0,Y 305.139,Z 1154.555,A -85,B 0,C 180,E1 15046.367,E2 15046.367} C_VEL
LIN {X 0,Y 304.357,Z 1159.417,A -85,B 0,C 180,E1 15042.522,E2 15042.522} C_VEL
LIN {X 0,Y 304.027,Z 1163.21,A -85,B 0,C 180,E1 15038.51,E2 15038.51} C_VEL
LIN {X 0,Y 303.958,Z 1165.432,A -85,B 0,C 180,E1 15034.528,E2 15034.528} C_VEL
LIN {X 0,Y 303.963,Z 1166.285,A -85,B 0,C 180,E1 15031.13,E2 15031.13} C_VEL
LIN {X 0,Y 303.953,Z 1166.092,A -85,B 0,C 180,E1 15027.36,E2 15027.36} C_VEL
LIN {X 0,Y 303.972,Z 1164.406,A -85,B 0,C 180,E1 15023.389,E2 15023.389} C_VEL
LIN {X 0,Y 304.09,Z 1161.883,A -85,B 0,C 180,E1 15019.964,E2 15019.964} C_VEL
LIN {X 0,Y 304.598,Z 1157.692,A -85,B 0,C 180,E1 15015.941,E2 15015.941} C_VEL
LIN {X 0,Y 305.68,Z 1151.859,A -85,B 0,C 180,E1 15011.896,E2 15011.896} C_VEL
LIN {X 0,Y 307.539,Z 1144.62,A -85,B 0,C 180,E1 15007.843,E2 15007.843} C_VEL
